KUKA KRL program: EPS_2_25252_SD5A_A_20250910061727.src

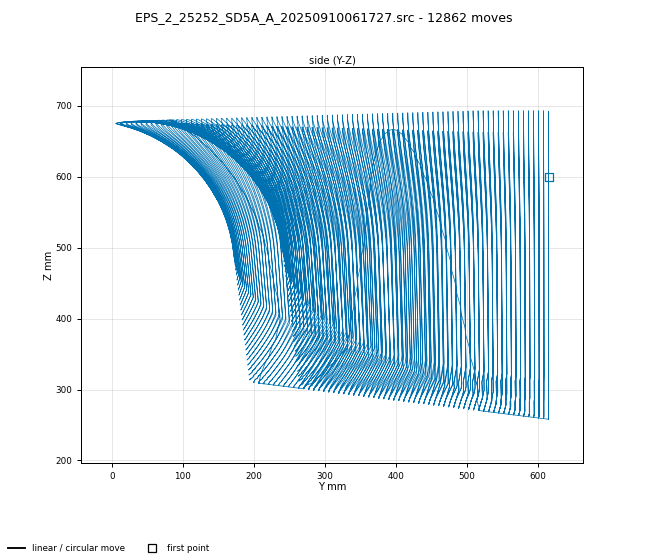
[picture p0: tool path of EPS_2_25252_SD5A_A_20250910061727.src, 12862 of 12864 moves have a stored position in this frame; points joined in program order, loops and branches not executed]
&ACCESS RVP
&REL 4
&COMMENT QRS 19112012
&PARAM EDITMASK = *
DEF PART()
EXT BAS (BAS_COMMAND :IN,REAL :IN )
INT I
BAS (#INITMOV,0 )

;KUKA QRS Post kuka4.cps  Date:22-06-2017 !

File_ID=2838

QRS_PRE_INIT()

;Init var - Until changes are made in qrs_pre_init
Outlet_Square_prg=0
Inlet_1_Square_prg=0
Inlet_2_Square_prg=0
Inlet_3_Square_prg=0
Inlet_4_Square_prg=0
Inlet_5_Square_prg=0

Outlet_1={X 0.000, Y 512.630, Z 510.000, B 0.000, E1 0.000 }
Inlet_1={X 0.000, Y 514.870, Z 480.000, B 0.000, E1 167.000 }
Outlet_1_type=366
Inlet_1_type=366
;QRS#1=Sidecore dimensions
;QRS#2=375-15" PVC SDR 35
;QRS#3=375-15" PVC SDR 35
;QRS#4=
;QRS#5=
;QRS#6=
;QRS#7=
;QRS#8=
;QRS#9=20Y PSX
;QRS#10=20Y PSX
;QRS#11=
;QRS#12=
;QRS#13=
;QRS#14=
;QRS#15=
;QRS#16=1220x127x991 3,25'
;QRS#17=EPS Height
;QRS#18=693
;QRS#19=*
;QRS#20= UPDATED VERSION 22-06-2017
;QRS#21=*
Outlet_Square=0250
Inlet_1_Square=0250
Inlet_2_Square=0
Inlet_3_Square=0
Inlet_4_Square=0
Inlet_5_Square=0
Mill_Square=1
Outlet_Square_Prg=252
Inlet_1_Square_prg=252

QRS_INIT()

$ADVANCE=5

; T1
PTP {E1 173.62,E2 173.62}
PTP {X 0,Y 615.5,A -85,B 0,C 180,E1 173.62,E2 173.62,E3 0,E4 0,E5 0,E6 0}
QRS_SPEED_INIT()
LIN {X 0,Y 615.5,Z 600,A -85,B 0,C 180,E1 173.62,E2 173.62,E3 0,E4 0,E5 0,E6 0} C_VEL
LIN {X 0,Y 615.5,Z 268.19,A -85,B 0,C 180,E1 173.62,E2 173.62} C_VEL
LIN {X 0,Y 615.5,Z 260.011,A -85,B 0,C 180,E1 173.62,E2 173.62} C_VEL
LIN {X 0,Y 615.475,Z 258.011,A -85,B 0,C 180,E1 173.434,E2 173.434} C_VEL
LIN {X 0,Y 615.437,Z 258.007,A -85,B 0,C 180,E1 170.8,E2 170.8} C_VEL
LIN {X 0,Y 615.481,Z 258.003,A -85,B 0,C 180,E1 168.139,E2 168.139} C_VEL
LIN {X 0,Y 615.462,Z 258.011,A -85,B 0,C 180,E1 165.45,E2 165.45} C_VEL
LIN {X 0,Y 615.455,Z 258.011,A -85,B 0,C 180,E1 163.412,E2 163.412} C_VEL
LIN {X 0,Y 615.445,Z 258.011,A -85,B 0,C 180,E1 161.352,E2 161.352} C_VEL
LIN {X 0,Y 615.436,Z 258.011,A -85,B 0,C 180,E1 159.267,E2 159.267} C_VEL
LIN {X 0,Y 615.426,Z 258.011,A -85,B 0,C 180,E1 157.153,E2 157.153} C_VEL
LIN {X 0,Y 615.418,Z 258.011,A -85,B 0,C 180,E1 155.005,E2 155.005} C_VEL
LIN {X 0,Y 615.418,Z 258.011,A -85,B 0,C 180,E1 152.819,E2 152.819} C_VEL
LIN {X 0,Y 615.467,Z 258.011,A -85,B 0,C 180,E1 150.209,E2 150.209} C_VEL
LIN {X 0,Y 615.438,Z 258.012,A -85,B 0,C 180,E1 147.539,E2 147.539} C_VEL
LIN {X 0,Y 615.413,Z 258.012,A -85,B 0,C 180,E1 145.18,E2 145.18} C_VEL
LIN {X 0,Y 615.42,Z 258.012,A -85,B 0,C 180,E1 142.753,E2 142.753} C_VEL
LIN {X 0,Y 615.486,Z 258.009,A -85,B 0,C 180,E1 139.911,E2 139.911} C_VEL
LIN {X 0,Y 615.451,Z 258.009,A -85,B 0,C 180,E1 137.643,E2 137.643} C_VEL
LIN {X 0,Y 615.422,Z 258.01,A -85,B 0,C 180,E1 135.075,E2 135.075} C_VEL
LIN {X 0,Y 615.425,Z 258.009,A -85,B 0,C 180,E1 133.04,E2 133.04} C_VEL
LIN {X 0,Y 615.45,Z 258.011,A -85,B 0,C 180,E1 130.61,E2 130.61} C_VEL
LIN {X 0,Y 615.454,Z 258.005,A -85,B 0,C 180,E1 127.628,E2 127.628} C_VEL
LIN {X 0,Y 615.432,Z 258.012,A -85,B 0,C 180,E1 127.246,E2 127.246} C_VEL
LIN {X 0,Y 615.457,Z 282.781,A -85,B 0,C 180,E1 124.979,E2 124.979} C_VEL
LIN {X 0,Y 615.491,Z 489.244,A -85,B 0,C 180,E1 122.426,E2 122.426} C_VEL
LIN {X 0,Y 615.493,Z 505.497,A -85,B 0,C 180,E1 122.088,E2 122.088} C_VEL
LIN {X 0,Y 615.497,Z 521.955,A -85,B 0,C 180,E1 121.61,E2 121.61} C_VEL
LIN {X 0,Y 615.49,Z 537.997,A -85,B 0,C 180,E1 121.002,E2 121.002} C_VEL
LIN {X 0,Y 615.49,Z 551.97,A -85,B 0,C 180,E1 120.349,E2 120.349} C_VEL
LIN {X 0,Y 615.498,Z 566.878,A -85,B 0,C 180,E1 119.503,E2 119.503} C_VEL
LIN {X 0,Y 615.494,Z 580.891,A -85,B 0,C 180,E1 118.554,E2 118.554} C_VEL
LIN {X 0,Y 615.493,Z 594.61,A -85,B 0,C 180,E1 117.453,E2 117.453} C_VEL
LIN {X 0,Y 615.494,Z 607.149,A -85,B 0,C 180,E1 116.261,E2 116.261} C_VEL
LIN {X 0,Y 615.496,Z 618.457,A -85,B 0,C 180,E1 114.992,E2 114.992} C_VEL
LIN {X 0,Y 615.493,Z 627.669,A -85,B 0,C 180,E1 113.782,E2 113.782} C_VEL
LIN {X 0,Y 615.491,Z 636.834,A -85,B 0,C 180,E1 112.346,E2 112.346} C_VEL
LIN {X 0,Y 615.491,Z 643.498,A -85,B 0,C 180,E1 111.081,E2 111.081} C_VEL
LIN {X 0,Y 615.491,Z 649.613,A -85,B 0,C 180,E1 109.685,E2 109.685} C_VEL
LIN {X 0,Y 615.486,Z 653.438,A -85,B 0,C 180,E1 108.603,E2 108.603} C_VEL
LIN {X 0,Y 615.483,Z 657.237,A -85,B 0,C 180,E1 107.271,E2 107.271} C_VEL
LIN {X 0,Y 615.491,Z 659.946,A -85,B 0,C 180,E1 105.905,E2 105.905} C_VEL
LIN {X 0,Y 615.493,Z 661.669,A -85,B 0,C 180,E1 104.549,E2 104.549} C_VEL
LIN {X 0,Y 615.485,Z 662.336,A -85,B 0,C 180,E1 103.201,E2 103.201} C_VEL
LIN {X 0,Y 615.493,Z 662.022,A -85,B 0,C 180,E1 101.861,E2 101.861} C_VEL
LIN {X 0,Y 615.489,Z 660.742,A -85,B 0,C 180,E1 100.527,E2 100.527} C_VEL
LIN {X 0,Y 615.492,Z 658.451,A -85,B 0,C 180,E1 99.199,E2 99.199} C_VEL
LIN {X 0,Y 615.496,Z 655.195,A -85,B 0,C 180,E1 97.876,E2 97.876} C_VEL
LIN {X 0,Y 615.488,Z 650.852,A -85,B 0,C 180,E1 96.557,E2 96.557} C_VEL
LIN {X 0,Y 615.492,Z 645.49,A -85,B 0,C 180,E1 95.241,E2 95.241} C_VEL
LIN {X 0,Y 615.488,Z 637.049,A -85,B 0,C 180,E1 93.601,E2 93.601} C_VEL
LIN {X 0,Y 615.488,Z 628.759,A -85,B 0,C 180,E1 92.291,E2 92.291} C_VEL
LIN {X 0,Y 615.493,Z 618.969,A -85,B 0,C 180,E1 90.981,E2 90.981} C_VEL
LIN {X 0,Y 615.491,Z 607.385,A -85,B 0,C 180,E1 89.673,E2 89.673} C_VEL
LIN {X 0,Y 615.494,Z 595.424,A -85,B 0,C 180,E1 88.528,E2 88.528} C_VEL
LIN {X 0,Y 615.496,Z 582.372,A -85,B 0,C 180,E1 87.464,E2 87.464} C_VEL
LIN {X 0,Y 615.498,Z 569.42,A -85,B 0,C 180,E1 86.563,E2 86.563} C_VEL
LIN {X 0,Y 615.498,Z 555.382,A -85,B 0,C 180,E1 85.744,E2 85.744} C_VEL
LIN {X 0,Y 615.498,Z 540.224,A -85,B 0,C 180,E1 85.005,E2 85.005} C_VEL
LIN {X 0,Y 615.498,Z 524.623,A -85,B 0,C 180,E1 84.389,E2 84.389} C_VEL
LIN {X 0,Y 615.497,Z 508.547,A -85,B 0,C 180,E1 83.896,E2 83.896} C_VEL
LIN {X 0,Y 615.489,Z 491.531,A -85,B 0,C 180,E1 83.526,E2 83.526} C_VEL
LIN {X 0,Y 615.495,Z 466.17,A -85,B 0,C 180,E1 83.185,E2 83.185} C_VEL
LIN {X 0,Y 615.461,Z 282.717,A -85,B 0,C 180,E1 80.925,E2 80.925} C_VEL
LIN {X 0,Y 615.44,Z 258.005,A -85,B 0,C 180,E1 78.66,E2 78.66} C_VEL
LIN {X 0,Y 615.49,Z 258.002,A -85,B 0,C 180,E1 76.068,E2 76.068} C_VEL
LIN {X 0,Y 615.462,Z 258.011,A -85,B 0,C 180,E1 73.413,E2 73.413} C_VEL
LIN {X 0,Y 615.453,Z 258.011,A -85,B 0,C 180,E1 71.353,E2 71.353} C_VEL
LIN {X 0,Y 615.443,Z 258.01,A -85,B 0,C 180,E1 69.268,E2 69.268} C_VEL
LIN {X 0,Y 615.434,Z 258.01,A -85,B 0,C 180,E1 67.153,E2 67.153} C_VEL
LIN {X 0,Y 615.426,Z 258.01,A -85,B 0,C 180,E1 65.006,E2 65.006} C_VEL
LIN {X 0,Y 615.424,Z 258.009,A -85,B 0,C 180,E1 62.82,E2 62.82} C_VEL
LIN {X 0,Y 615.469,Z 258.008,A -85,B 0,C 180,E1 60.209,E2 60.209} C_VEL
LIN {X 0,Y 615.45,Z 258.012,A -85,B 0,C 180,E1 57.54,E2 57.54} C_VEL
LIN {X 0,Y 615.418,Z 258.012,A -85,B 0,C 180,E1 55.18,E2 55.18} C_VEL
LIN {X 0,Y 615.417,Z 258.012,A -85,B 0,C 180,E1 52.753,E2 52.753} C_VEL
LIN {X 0,Y 615.488,Z 258.012,A -85,B 0,C 180,E1 49.912,E2 49.912} C_VEL
LIN {X 0,Y 615.447,Z 258.012,A -85,B 0,C 180,E1 47.644,E2 47.644} C_VEL
LIN {X 0,Y 615.413,Z 258.012,A -85,B 0,C 180,E1 45.076,E2 45.076} C_VEL
LIN {X 0,Y 615.414,Z 258.011,A -85,B 0,C 180,E1 43.04,E2 43.04} C_VEL
LIN {X 0,Y 615.417,Z 258.011,A -85,B 0,C 180,E1 41.087,E2 41.087} C_VEL
LIN {X 0,Y 615.421,Z 258.011,A -85,B 0,C 180,E1 38.91,E2 38.91} C_VEL
LIN {X 0,Y 615.459,Z 258.012,A -85,B 0,C 180,E1 36.427,E2 36.427} C_VEL
LIN {X 0,Y 615.442,Z 258.008,A -85,B 0,C 180,E1 33.528,E2 33.528} C_VEL
LIN {X 0,Y 615.427,Z 258.009,A -85,B 0,C 180,E1 31.077,E2 31.077} C_VEL
LIN {X 0,Y 615.445,Z 258.011,A -85,B 0,C 180,E1 28.661,E2 28.661} C_VEL
LIN {X 0,Y 615.463,Z 258.004,A -85,B 0,C 180,E1 25.717,E2 25.717} C_VEL
LIN {X 0,Y 615.449,Z 258.005,A -85,B 0,C 180,E1 23.558,E2 23.558} C_VEL
LIN {X 0,Y 615.443,Z 258.005,A -85,B 0,C 180,E1 21.434,E2 21.434} C_VEL
LIN {X 0,Y 615.44,Z 258.005,A -85,B 0,C 180,E1 19.34,E2 19.34} C_VEL
LIN {X 0,Y 615.44,Z 258.006,A -85,B 0,C 180,E1 17.272,E2 17.272} C_VEL
LIN {X 0,Y 615.482,Z 258.011,A -85,B 0,C 180,E1 14.55,E2 14.55} C_VEL
LIN {X 0,Y 615.482,Z 258,A -85,B 0,C 180,E1 11.861,E2 11.861} C_VEL
LIN {X 0,Y 615.447,Z 258.006,A -85,B 0,C 180,E1 9.2,E2 9.2} C_VEL
LIN {X 0,Y 615.491,Z 258.013,A -85,B 0,C 180,E1 6.557,E2 6.557} C_VEL
LIN {X 0,Y 615.484,Z 257.999,A -85,B 0,C 180,E1 3.929,E2 3.929} C_VEL
LIN {X 0,Y 615.453,Z 258.004,A -85,B 0,C 180,E1 1.309,E2 1.309} C_VEL
LIN {X 0,Y 615.489,Z 258.011,A -85,B 0,C 180,E1 -1.308,E2 -1.308} C_VEL
LIN {X 0,Y 615.49,Z 257.998,A -85,B 0,C 180,E1 -3.928,E2 -3.928} C_VEL
LIN {X 0,Y 615.46,Z 258.002,A -85,B 0,C 180,E1 -6.557,E2 -6.557} C_VEL
LIN {X 0,Y 615.488,Z 258.011,A -85,B 0,C 180,E1 -9.198,E2 -9.198} C_VEL
LIN {X 0,Y 615.493,Z 257.997,A -85,B 0,C 180,E1 -11.86,E2 -11.86} C_VEL
LIN {X 0,Y 615.465,Z 258.002,A -85,B 0,C 180,E1 -14.549,E2 -14.549} C_VEL
LIN {X 0,Y 615.493,Z 258.012,A -85,B 0,C 180,E1 -17.27,E2 -17.27} C_VEL
LIN {X 0,Y 615.488,Z 257.995,A -85,B 0,C 180,E1 -20.032,E2 -20.032} C_VEL
LIN {X 0,Y 615.477,Z 258.007,A -85,B 0,C 180,E1 -22.845,E2 -22.845} C_VEL
LIN {X 0,Y 615.481,Z 257.999,A -85,B 0,C 180,E1 -25.716,E2 -25.716} C_VEL
LIN {X 0,Y 615.474,Z 258.001,A -85,B 0,C 180,E1 -28.448,E2 -28.448} C_VEL
LIN {X 0,Y 615.484,Z 258.015,A -85,B 0,C 180,E1 -31.085,E2 -31.085} C_VEL
LIN {X 0,Y 615.493,Z 257.993,A -85,B 0,C 180,E1 -34.021,E2 -34.021} C_VEL
LIN {X 0,Y 615.488,Z 258.014,A -85,B 0,C 180,E1 -36.937,E2 -36.937} C_VEL
LIN {X 0,Y 615.478,Z 257.998,A -85,B 0,C 180,E1 -39.751,E2 -39.751} C_VEL
LIN {X 0,Y 615.482,Z 258,A -85,B 0,C 180,E1 -42.353,E2 -42.353} C_VEL
LIN {X 0,Y 615.484,Z 258.009,A -85,B 0,C 180,E1 -45.069,E2 -45.069} C_VEL
LIN {X 0,Y 615.489,Z 257.995,A -85,B 0,C 180,E1 -47.919,E2 -47.919} C_VEL
LIN {X 0,Y 615.487,Z 258.01,A -85,B 0,C 180,E1 -50.938,E2 -50.938} C_VEL
LIN {X 0,Y 615.469,Z 258,A -85,B 0,C 180,E1 -53.574,E2 -53.574} C_VEL
LIN {X 0,Y 615.488,Z 258.006,A -85,B 0,C 180,E1 -56.465,E2 -56.465} C_VEL
LIN {X 0,Y 615.469,Z 258.007,A -85,B 0,C 180,E1 -59.079,E2 -59.079} C_VEL
LIN {X 0,Y 615.464,Z 258,A -85,B 0,C 180,E1 -61.553,E2 -61.553} C_VEL
LIN {X 0,Y 615.465,Z 258.184,A -85,B 0,C 180,E1 -63.601,E2 -63.601} C_VEL
LIN {X 0,Y 615.476,Z 290.167,A -85,B 0,C 180,E1 -66.217,E2 -66.217} C_VEL
LIN {X 0,Y 615.493,Z 312.012,A -85,B 0,C 180,E1 -67.974,E2 -67.974} C_VEL
LIN {X 0,Y 615.491,Z 519.433,A -85,B 0,C 180,E1 -70.532,E2 -70.532} C_VEL
LIN {X 0,Y 615.493,Z 535.998,A -85,B 0,C 180,E1 -70.879,E2 -70.879} C_VEL
LIN {X 0,Y 615.493,Z 550.934,A -85,B 0,C 180,E1 -71.311,E2 -71.311} C_VEL
LIN {X 0,Y 615.491,Z 566.349,A -85,B 0,C 180,E1 -71.881,E2 -71.881} C_VEL
LIN {X 0,Y 615.493,Z 581.006,A -85,B 0,C 180,E1 -72.558,E2 -72.558} C_VEL
LIN {X 0,Y 615.5,Z 594.837,A -85,B 0,C 180,E1 -73.328,E2 -73.328} C_VEL
LIN {X 0,Y 615.499,Z 609.038,A -85,B 0,C 180,E1 -74.265,E2 -74.265} C_VEL
LIN {X 0,Y 615.495,Z 622.093,A -85,B 0,C 180,E1 -75.282,E2 -75.282} C_VEL
LIN {X 0,Y 615.494,Z 633.214,A -85,B 0,C 180,E1 -76.294,E2 -76.294} C_VEL
LIN {X 0,Y 615.493,Z 644.291,A -85,B 0,C 180,E1 -77.47,E2 -77.47} C_VEL
LIN {X 0,Y 615.494,Z 653.767,A -85,B 0,C 180,E1 -78.64,E2 -78.64} C_VEL
LIN {X 0,Y 615.496,Z 662.964,A -85,B 0,C 180,E1 -79.972,E2 -79.972} C_VEL
LIN {X 0,Y 615.489,Z 671.502,A -85,B 0,C 180,E1 -81.463,E2 -81.463} C_VEL
LIN {X 0,Y 615.491,Z 678.982,A -85,B 0,C 180,E1 -83.102,E2 -83.102} C_VEL
LIN {X 0,Y 615.492,Z 684.741,A -85,B 0,C 180,E1 -84.759,E2 -84.759} C_VEL
LIN {X 0,Y 615.494,Z 688.076,A -85,B 0,C 180,E1 -86.072,E2 -86.072} C_VEL
LIN {X 0,Y 615.485,Z 690.504,A -85,B 0,C 180,E1 -87.382,E2 -87.382} C_VEL
LIN {X 0,Y 615.488,Z 691.87,A -85,B 0,C 180,E1 -88.691,E2 -88.691} C_VEL
LIN {X 0,Y 615.489,Z 692.39,A -85,B 0,C 180,E1 -90,E2 -90} C_VEL
LIN {X 0,Y 615.488,Z 691.87,A -85,B 0,C 180,E1 -91.309,E2 -91.309} C_VEL
LIN {X 0,Y 615.485,Z 690.504,A -85,B 0,C 180,E1 -92.618,E2 -92.618} C_VEL
LIN {X 0,Y 615.494,Z 688.076,A -85,B 0,C 180,E1 -93.929,E2 -93.929} C_VEL
LIN {X 0,Y 615.492,Z 684.741,A -85,B 0,C 180,E1 -95.241,E2 -95.241} C_VEL
LIN {X 0,Y 615.491,Z 678.982,A -85,B 0,C 180,E1 -96.898,E2 -96.898} C_VEL
LIN {X 0,Y 615.489,Z 671.501,A -85,B 0,C 180,E1 -98.537,E2 -98.537} C_VEL
LIN {X 0,Y 615.496,Z 662.963,A -85,B 0,C 180,E1 -100.028,E2 -100.028} C_VEL
LIN {X 0,Y 615.494,Z 653.765,A -85,B 0,C 180,E1 -101.36,E2 -101.36} C_VEL
LIN {X 0,Y 615.495,Z 644.29,A -85,B 0,C 180,E1 -102.53,E2 -102.53} C_VEL
LIN {X 0,Y 615.494,Z 633.212,A -85,B 0,C 180,E1 -103.706,E2 -103.706} C_VEL
LIN {X 0,Y 615.495,Z 621.113,A -85,B 0,C 180,E1 -104.803,E2 -104.803} C_VEL
LIN {X 0,Y 615.498,Z 606.706,A -85,B 0,C 180,E1 -105.905,E2 -105.905} C_VEL
LIN {X 0,Y 615.497,Z 592.012,A -85,B 0,C 180,E1 -106.843,E2 -106.843} C_VEL
LIN {X 0,Y 615.49,Z 577.507,A -85,B 0,C 180,E1 -107.613,E2 -107.613} C_VEL
LIN {X 0,Y 615.49,Z 562.245,A -85,B 0,C 180,E1 -108.282,E2 -108.282} C_VEL
LIN {X 0,Y 615.49,Z 546.989,A -85,B 0,C 180,E1 -108.819,E2 -108.819} C_VEL
LIN {X 0,Y 615.497,Z 530.513,A -85,B 0,C 180,E1 -109.251,E2 -109.251} C_VEL
LIN {X 0,Y 615.49,Z 514.919,A -85,B 0,C 180,E1 -109.533,E2 -109.533} C_VEL
LIN {X 0,Y 615.493,Z 312.01,A -85,B 0,C 180,E1 -112.026,E2 -112.026} C_VEL
LIN {X 0,Y 615.458,Z 276.401,A -85,B 0,C 180,E1 -114.903,E2 -114.903} C_VEL
LIN {X 0,Y 615.464,Z 258,A -85,B 0,C 180,E1 -116.422,E2 -116.422} C_VEL
LIN {X 0,Y 615.461,Z 258.003,A -85,B 0,C 180,E1 -118.66,E2 -118.66} C_VEL
LIN {X 0,Y 615.481,Z 258.01,A -85,B 0,C 180,E1 -121.085,E2 -121.085} C_VEL
LIN {X 0,Y 615.493,Z 257.995,A -85,B 0,C 180,E1 -124.022,E2 -124.022} C_VEL
LIN {X 0,Y 615.478,Z 258.008,A -85,B 0,C 180,E1 -126.936,E2 -126.936} C_VEL
LIN {X 0,Y 615.483,Z 257.999,A -85,B 0,C 180,E1 -129.751,E2 -129.751} C_VEL
LIN {X 0,Y 615.475,Z 257.999,A -85,B 0,C 180,E1 -132.354,E2 -132.354} C_VEL
LIN {X 0,Y 615.493,Z 258.014,A -85,B 0,C 180,E1 -135.068,E2 -135.068} C_VEL
LIN {X 0,Y 615.49,Z 257.995,A -85,B 0,C 180,E1 -137.92,E2 -137.92} C_VEL
LIN {X 0,Y 615.482,Z 257.997,A -85,B 0,C 180,E1 -140.25,E2 -140.25} C_VEL
LIN {X 0,Y 615.491,Z 258.011,A -85,B 0,C 180,E1 -143.063,E2 -143.063} C_VEL
LIN {X 0,Y 615.491,Z 257.994,A -85,B 0,C 180,E1 -145.979,E2 -145.979} C_VEL
LIN {X 0,Y 615.486,Z 258.015,A -85,B 0,C 180,E1 -148.915,E2 -148.915} C_VEL
LIN {X 0,Y 615.471,Z 258,A -85,B 0,C 180,E1 -151.553,E2 -151.553} C_VEL
LIN {X 0,Y 615.486,Z 258,A -85,B 0,C 180,E1 -154.285,E2 -154.285} C_VEL
LIN {X 0,Y 615.486,Z 258.004,A -85,B 0,C 180,E1 -156.444,E2 -156.444} C_VEL
LIN {X 0,Y 615.465,Z 258.005,A -85,B 0,C 180,E1 -159.269,E2 -159.269} C_VEL
LIN {X 0,Y 615.493,Z 257.996,A -85,B 0,C 180,E1 -162.044,E2 -162.044} C_VEL
LIN {X 0,Y 615.484,Z 258.012,A -85,B 0,C 180,E1 -164.774,E2 -164.774} C_VEL
LIN {X 0,Y 615.459,Z 258.002,A -85,B 0,C 180,E1 -167.47,E2 -167.47} C_VEL
LIN {X 0,Y 615.493,Z 258,A -85,B 0,C 180,E1 -170.138,E2 -170.138} C_VEL
LIN {X 0,Y 615.474,Z 258.01,A -85,B 0,C 180,E1 -172.785,E2 -172.785} C_VEL
LIN {X 0,Y 615.452,Z 258.003,A -85,B 0,C 180,E1 -175.416,E2 -175.416} C_VEL
LIN {X 0,Y 615.498,Z 257.999,A -85,B 0,C 180,E1 -178.037,E2 -178.037} C_VEL
LIN {X 0,Y 615.474,Z 258.011,A -85,B 0,C 180,E1 -180.655,E2 -180.655} C_VEL
LIN {X 0,Y 615.443,Z 258.005,A -85,B 0,C 180,E1 -183.274,E2 -183.274} C_VEL
LIN {X 0,Y 615.485,Z 258.001,A -85,B 0,C 180,E1 -185.899,E2 -185.899} C_VEL
LIN {X 0,Y 615.475,Z 258.011,A -85,B 0,C 180,E1 -186.566,E2 -186.566} C_VEL
LIN {X 0,Y 614.772,Z 258.153,A -85,B 0,C 180,E1 -187.112,E2 -187.112} C_VEL
LIN {X 0,Y 611.917,Z 258.573,A -85,B 0,C 180,E1 -187.998,E2 -187.998} C_VEL
LIN {X 0,Y 609.53,Z 258.879,A -85,B 0,C 180,E1 -188.711,E2 -188.711} C_VEL
LIN {X 0,Y 608.51,Z 258.994,A -85,B 0,C 180,E1 -189.26,E2 -189.26} C_VEL
LIN {X 0,Y 608.428,Z 259.003,A -85,B 0,C 180,E1 -189.446,E2 -189.446} C_VEL
LIN {X 0,Y 608.455,Z 259.005,A -85,B 0,C 180,E1 -192,E2 -192} C_VEL
LIN {X 0,Y 608.417,Z 259.007,A -85,B 0,C 180,E1 -194.722,E2 -194.722} C_VEL
LIN {X 0,Y 608.419,Z 259.006,A -85,B 0,C 180,E1 -196.785,E2 -196.785} C_VEL
LIN {X 0,Y 608.421,Z 259.005,A -85,B 0,C 180,E1 -199.572,E2 -199.572} C_VEL
LIN {X 0,Y 608.433,Z 259.007,A -85,B 0,C 180,E1 -202.47,E2 -202.47} C_VEL
LIN {X 0,Y 608.424,Z 259.007,A -85,B 0,C 180,E1 -204.573,E2 -204.573} C_VEL
LIN {X 0,Y 608.403,Z 259.006,A -85,B 0,C 180,E1 -207.193,E2 -207.193} C_VEL
LIN {X 0,Y 608.455,Z 259.009,A -85,B 0,C 180,E1 -209.969,E2 -209.969} C_VEL
LIN {X 0,Y 608.407,Z 259.006,A -85,B 0,C 180,E1 -212.883,E2 -212.883} C_VEL
LIN {X 0,Y 608.398,Z 259.008,A -85,B 0,C 180,E1 -215.281,E2 -215.281} C_VEL
LIN {X 0,Y 608.423,Z 259.009,A -85,B 0,C 180,E1 -218.235,E2 -218.235} C_VEL
LIN {X 0,Y 608.437,Z 259.006,A -85,B 0,C 180,E1 -220.327,E2 -220.327} C_VEL
LIN {X 0,Y 608.425,Z 259.007,A -85,B 0,C 180,E1 -222.33,E2 -222.33} C_VEL
LIN {X 0,Y 608.404,Z 259.006,A -85,B 0,C 180,E1 -224.801,E2 -224.801} C_VEL
LIN {X 0,Y 608.397,Z 259.007,A -85,B 0,C 180,E1 -227.035,E2 -227.035} C_VEL
LIN {X 0,Y 608.399,Z 259.007,A -85,B 0,C 180,E1 -228.819,E2 -228.819} C_VEL
LIN {X 0,Y 608.41,Z 259.01,A -85,B 0,C 180,E1 -231.407,E2 -231.407} C_VEL
LIN {X 0,Y 608.448,Z 259.144,A -85,B 0,C 180,E1 -232.562,E2 -232.562} C_VEL
LIN {X 0,Y 608.699,Z 265.928,A -85,B 0,C 180,E1 -233.206,E2 -233.206} C_VEL
LIN {X 0,Y 608.688,Z 283.12,A -85,B 0,C 180,E1 -234.776,E2 -234.776} C_VEL
LIN {X 0,Y 608.886,Z 299.347,A -85,B 0,C 180,E1 -234.986,E2 -234.986} C_VEL
LIN {X 0,Y 608.795,Z 489.212,A -85,B 0,C 180,E1 -237.351,E2 -237.351} C_VEL
LIN {X 0,Y 608.774,Z 505.767,A -85,B 0,C 180,E1 -237.699,E2 -237.699} C_VEL
LIN {X 0,Y 608.739,Z 521.663,A -85,B 0,C 180,E1 -238.165,E2 -238.165} C_VEL
LIN {X 0,Y 608.695,Z 537.166,A -85,B 0,C 180,E1 -238.752,E2 -238.752} C_VEL
LIN {X 0,Y 608.651,Z 552.299,A -85,B 0,C 180,E1 -239.465,E2 -239.465} C_VEL
LIN {X 0,Y 608.632,Z 567.204,A -85,B 0,C 180,E1 -240.324,E2 -240.324} C_VEL
LIN {X 0,Y 608.591,Z 580.323,A -85,B 0,C 180,E1 -241.221,E2 -241.221} C_VEL
LIN {X 0,Y 608.545,Z 593.768,A -85,B 0,C 180,E1 -242.3,E2 -242.3} C_VEL
LIN {X 0,Y 608.523,Z 605.625,A -85,B 0,C 180,E1 -243.414,E2 -243.414} C_VEL
LIN {X 0,Y 608.478,Z 616.052,A -85,B 0,C 180,E1 -244.554,E2 -244.554} C_VEL
LIN {X 0,Y 608.477,Z 626.718,A -85,B 0,C 180,E1 -245.927,E2 -245.927} C_VEL
LIN {X 0,Y 608.464,Z 635.273,A -85,B 0,C 180,E1 -247.236,E2 -247.236} C_VEL
LIN {X 0,Y 608.455,Z 643.098,A -85,B 0,C 180,E1 -248.663,E2 -248.663} C_VEL
LIN {X 0,Y 608.433,Z 649.462,A -85,B 0,C 180,E1 -250.077,E2 -250.077} C_VEL
LIN {X 0,Y 608.423,Z 653.828,A -85,B 0,C 180,E1 -251.299,E2 -251.299} C_VEL
LIN {X 0,Y 608.41,Z 657.363,A -85,B 0,C 180,E1 -252.522,E2 -252.522} C_VEL
LIN {X 0,Y 608.428,Z 660.267,A -85,B 0,C 180,E1 -253.905,E2 -253.905} C_VEL
LIN {X 0,Y 608.416,Z 662.146,A -85,B 0,C 180,E1 -255.278,E2 -255.278} C_VEL
LIN {X 0,Y 608.431,Z 662.911,A -85,B 0,C 180,E1 -256.643,E2 -256.643} C_VEL
LIN {X 0,Y 608.437,Z 662.738,A -85,B 0,C 180,E1 -258,E2 -258} C_VEL
LIN {X 0,Y 608.43,Z 661.512,A -85,B 0,C 180,E1 -259.349,E2 -259.349} C_VEL
LIN {X 0,Y 608.419,Z 659.338,A -85,B 0,C 180,E1 -260.693,E2 -260.693} C_VEL
LIN {X 0,Y 608.42,Z 656.121,A -85,B 0,C 180,E1 -262.032,E2 -262.032} C_VEL
LIN {X 0,Y 608.448,Z 651.761,A -85,B 0,C 180,E1 -263.397,E2 -263.397} C_VEL
LIN {X 0,Y 608.456,Z 646.54,A -85,B 0,C 180,E1 -264.698,E2 -264.698} C_VEL
LIN {X 0,Y 608.434,Z 639.993,A -85,B 0,C 180,E1 -266.026,E2 -266.026} C_VEL
LIN {X 0,Y 608.46,Z 632.217,A -85,B 0,C 180,E1 -267.352,E2 -267.352} C_VEL
LIN {X 0,Y 608.478,Z 622.95,A -85,B 0,C 180,E1 -268.676,E2 -268.676} C_VEL
LIN {X 0,Y 608.486,Z 611.978,A -85,B 0,C 180,E1 -270,E2 -270} C_VEL
LIN {X 0,Y 608.519,Z 600.706,A -85,B 0,C 180,E1 -271.158,E2 -271.158} C_VEL
LIN {X 0,Y 608.558,Z 587.484,A -85,B 0,C 180,E1 -272.316,E2 -272.316} C_VEL
LIN {X 0,Y 608.612,Z 574.126,A -85,B 0,C 180,E1 -273.31,E2 -273.31} C_VEL
LIN {X 0,Y 608.638,Z 559.633,A -85,B 0,C 180,E1 -274.221,E2 -274.221} C_VEL
LIN {X 0,Y 608.673,Z 545.387,A -85,B 0,C 180,E1 -274.968,E2 -274.968} C_VEL
LIN {X 0,Y 608.73,Z 529.827,A -85,B 0,C 180,E1 -275.632,E2 -275.632} C_VEL
LIN {X 0,Y 608.763,Z 513.799,A -85,B 0,C 180,E1 -276.172,E2 -276.172} C_VEL
LIN {X 0,Y 608.789,Z 497.872,A -85,B 0,C 180,E1 -276.575,E2 -276.575} C_VEL
LIN {X 0,Y 608.805,Z 481.487,A -85,B 0,C 180,E1 -276.851,E2 -276.851} C_VEL
LIN {X 0,Y 608.878,Z 285.382,A -85,B 0,C 180,E1 -279.279,E2 -279.279} C_VEL
LIN {X 0,Y 608.668,Z 282.6,A -85,B 0,C 180,E1 -279.345,E2 -279.345} C_VEL
LIN {X 0,Y 608.696,Z 261.258,A -85,B 0,C 180,E1 -281.32,E2 -281.32} C_VEL
LIN {X 0,Y 608.442,Z 259.004,A -85,B 0,C 180,E1 -281.556,E2 -281.556} C_VEL
LIN {X 0,Y 608.475,Z 259.003,A -85,B 0,C 180,E1 -284.037,E2 -284.037} C_VEL
LIN {X 0,Y 608.424,Z 259.006,A -85,B 0,C 180,E1 -286.785,E2 -286.785} C_VEL
LIN {X 0,Y 608.424,Z 259.005,A -85,B 0,C 180,E1 -289.571,E2 -289.571} C_VEL
LIN {X 0,Y 608.439,Z 259.009,A -85,B 0,C 180,E1 -292.407,E2 -292.407} C_VEL
LIN {X 0,Y 608.43,Z 259.007,A -85,B 0,C 180,E1 -294.572,E2 -294.572} C_VEL
LIN {X 0,Y 608.408,Z 259.005,A -85,B 0,C 180,E1 -297.193,E2 -297.193} C_VEL
LIN {X 0,Y 608.46,Z 259.007,A -85,B 0,C 180,E1 -299.969,E2 -299.969} C_VEL
LIN {X 0,Y 608.414,Z 259.005,A -85,B 0,C 180,E1 -302.882,E2 -302.882} C_VEL
LIN {X 0,Y 608.399,Z 259.007,A -85,B 0,C 180,E1 -305.281,E2 -305.281} C_VEL
LIN {X 0,Y 608.424,Z 259.01,A -85,B 0,C 180,E1 -308.234,E2 -308.234} C_VEL
LIN {X 0,Y 608.436,Z 259.007,A -85,B 0,C 180,E1 -310.327,E2 -310.327} C_VEL
LIN {X 0,Y 608.421,Z 259.008,A -85,B 0,C 180,E1 -312.329,E2 -312.329} C_VEL
LIN {X 0,Y 608.396,Z 259.007,A -85,B 0,C 180,E1 -314.801,E2 -314.801} C_VEL
LIN {X 0,Y 608.387,Z 259.008,A -85,B 0,C 180,E1 -317.034,E2 -317.034} C_VEL
LIN {X 0,Y 608.389,Z 259.008,A -85,B 0,C 180,E1 -318.817,E2 -318.817} C_VEL
LIN {X 0,Y 608.404,Z 259.006,A -85,B 0,C 180,E1 -320.71,E2 -320.71} C_VEL
LIN {X 0,Y 608.394,Z 259.007,A -85,B 0,C 180,E1 -323.08,E2 -323.08} C_VEL
LIN {X 0,Y 608.441,Z 259.006,A -85,B 0,C 180,E1 -325.528,E2 -325.528} C_VEL
LIN {X 0,Y 608.455,Z 259.008,A -85,B 0,C 180,E1 -327.904,E2 -327.904} C_VEL
LIN {X 0,Y 608.456,Z 259.002,A -85,B 0,C 180,E1 -330.219,E2 -330.219} C_VEL
LIN {X 0,Y 608.412,Z 259.005,A -85,B 0,C 180,E1 -332.805,E2 -332.805} C_VEL
LIN {X 0,Y 608.436,Z 259.008,A -85,B 0,C 180,E1 -335.428,E2 -335.428} C_VEL
LIN {X 0,Y 608.448,Z 259.002,A -85,B 0,C 180,E1 -338.307,E2 -338.307} C_VEL
LIN {X 0,Y 608.439,Z 259.004,A -85,B 0,C 180,E1 -341.129,E2 -341.129} C_VEL
LIN {X 0,Y 608.46,Z 259.004,A -85,B 0,C 180,E1 -343.906,E2 -343.906} C_VEL
LIN {X 0,Y 608.433,Z 259.002,A -85,B 0,C 180,E1 -346.642,E2 -346.642} C_VEL
LIN {X 0,Y 608.456,Z 259.006,A -85,B 0,C 180,E1 -349.35,E2 -349.35} C_VEL
LIN {X 0,Y 608.475,Z 259,A -85,B 0,C 180,E1 -352.033,E2 -352.033} C_VEL
LIN {X 0,Y 608.435,Z 259.002,A -85,B 0,C 180,E1 -354.697,E2 -354.697} C_VEL
LIN {X 0,Y 608.481,Z 259.005,A -85,B 0,C 180,E1 -357.352,E2 -357.352} C_VEL
LIN {X 0,Y 608.477,Z 258.998,A -85,B 0,C 180,E1 -360,E2 -360} C_VEL
LIN {X 0,Y 608.451,Z 259.001,A -85,B 0,C 180,E1 -362.648,E2 -362.648} C_VEL
LIN {X 0,Y 608.468,Z 259.008,A -85,B 0,C 180,E1 -365.301,E2 -365.301} C_VEL
LIN {X 0,Y 608.479,Z 258.998,A -85,B 0,C 180,E1 -367.967,E2 -367.967} C_VEL
LIN {X 0,Y 608.444,Z 259.002,A -85,B 0,C 180,E1 -370.65,E2 -370.65} C_VEL
LIN {X 0,Y 608.471,Z 259.007,A -85,B 0,C 180,E1 -373.356,E2 -373.356} C_VEL
LIN {X 0,Y 608.457,Z 258.999,A -85,B 0,C 180,E1 -376.094,E2 -376.094} C_VEL
LIN {X 0,Y 608.449,Z 259.005,A -85,B 0,C 180,E1 -378.869,E2 -378.869} C_VEL
LIN {X 0,Y 608.467,Z 259,A -85,B 0,C 180,E1 -381.691,E2 -381.691} C_VEL
LIN {X 0,Y 608.451,Z 259.002,A -85,B 0,C 180,E1 -384.571,E2 -384.571} C_VEL
LIN {X 0,Y 608.483,Z 259.005,A -85,B 0,C 180,E1 -387.208,E2 -387.208} C_VEL
LIN {X 0,Y 608.468,Z 258.998,A -85,B 0,C 180,E1 -389.971,E2 -389.971} C_VEL
LIN {X 0,Y 608.451,Z 259.008,A -85,B 0,C 180,E1 -392.88,E2 -392.88} C_VEL
LIN {X 0,Y 608.439,Z 259.007,A -85,B 0,C 180,E1 -395.278,E2 -395.278} C_VEL
LIN {X 0,Y 608.467,Z 258.998,A -85,B 0,C 180,E1 -397.746,E2 -397.746} C_VEL
LIN {X 0,Y 608.454,Z 259.001,A -85,B 0,C 180,E1 -400.329,E2 -400.329} C_VEL
LIN {X 0,Y 608.453,Z 259.01,A -85,B 0,C 180,E1 -402.959,E2 -402.959} C_VEL
LIN {X 0,Y 608.456,Z 259,A -85,B 0,C 180,E1 -405.736,E2 -405.736} C_VEL
LIN {X 0,Y 608.461,Z 259.006,A -85,B 0,C 180,E1 -408.658,E2 -408.658} C_VEL
LIN {X 0,Y 608.462,Z 259,A -85,B 0,C 180,E1 -411.412,E2 -411.412} C_VEL
LIN {X 0,Y 608.46,Z 258.999,A -85,B 0,C 180,E1 -413.952,E2 -413.952} C_VEL
LIN {X 0,Y 608.466,Z 259.002,A -85,B 0,C 180,E1 -416.329,E2 -416.329} C_VEL
LIN {X 0,Y 608.459,Z 259.01,A -85,B 0,C 180,E1 -418.73,E2 -418.73} C_VEL
LIN {X 0,Y 608.453,Z 259.001,A -85,B 0,C 180,E1 -421.383,E2 -421.383} C_VEL
LIN {X 0,Y 608.449,Z 259.012,A -85,B 0,C 180,E1 -423.342,E2 -423.342} C_VEL
LIN {X 0,Y 608.824,Z 262.049,A -85,B 0,C 180,E1 -423.613,E2 -423.613} C_VEL
LIN {X 0,Y 608.729,Z 296.278,A -85,B 0,C 180,E1 -426.437,E2 -426.437} C_VEL
LIN {X 0,Y 608.713,Z 312.012,A -85,B 0,C 180,E1 -427.716,E2 -427.716} C_VEL
LIN {X 0,Y 608.9,Z 322.557,A -85,B 0,C 180,E1 -427.857,E2 -427.857} C_VEL
LIN {X 0,Y 608.795,Z 517.942,A -85,B 0,C 180,E1 -430.287,E2 -430.287} C_VEL
LIN {X 0,Y 608.796,Z 534.173,A -85,B 0,C 180,E1 -430.616,E2 -430.616} C_VEL
LIN {X 0,Y 608.737,Z 549.644,A -85,B 0,C 180,E1 -431.052,E2 -431.052} C_VEL
LIN {X 0,Y 608.711,Z 564.369,A -85,B 0,C 180,E1 -431.589,E2 -431.589} C_VEL
LIN {X 0,Y 608.678,Z 579.262,A -85,B 0,C 180,E1 -432.27,E2 -432.27} C_VEL
LIN {X 0,Y 608.616,Z 594.84,A -85,B 0,C 180,E1 -433.134,E2 -433.134} C_VEL
LIN {X 0,Y 608.579,Z 609.047,A -85,B 0,C 180,E1 -434.082,E2 -434.082} C_VEL
LIN {X 0,Y 608.556,Z 622.128,A -85,B 0,C 180,E1 -435.11,E2 -435.11} C_VEL
LIN {X 0,Y 608.528,Z 634.009,A -85,B 0,C 180,E1 -436.204,E2 -436.204} C_VEL
LIN {X 0,Y 608.49,Z 645.912,A -85,B 0,C 180,E1 -437.493,E2 -437.493} C_VEL
LIN {X 0,Y 608.487,Z 655.207,A -85,B 0,C 180,E1 -438.676,E2 -438.676} C_VEL
LIN {X 0,Y 608.471,Z 664.258,A -85,B 0,C 180,E1 -440.023,E2 -440.023} C_VEL
LIN {X 0,Y 608.444,Z 671.858,A -85,B 0,C 180,E1 -441.364,E2 -441.364} C_VEL
LIN {X 0,Y 608.437,Z 679.469,A -85,B 0,C 180,E1 -443.034,E2 -443.034} C_VEL
LIN {X 0,Y 608.435,Z 685.245,A -85,B 0,C 180,E1 -444.698,E2 -444.698} C_VEL
LIN {X 0,Y 608.431,Z 688.633,A -85,B 0,C 180,E1 -446.026,E2 -446.026} C_VEL
LIN {X 0,Y 608.412,Z 691.086,A -85,B 0,C 180,E1 -447.352,E2 -447.352} C_VEL
LIN {X 0,Y 608.441,Z 692.477,A -85,B 0,C 180,E1 -448.676,E2 -448.676} C_VEL
LIN {X 0,Y 608.429,Z 693,A -85,B 0,C 180,E1 -450,E2 -450} C_VEL
LIN {X 0,Y 608.441,Z 692.477,A -85,B 0,C 180,E1 -451.324,E2 -451.324} C_VEL
LIN {X 0,Y 608.412,Z 691.086,A -85,B 0,C 180,E1 -452.648,E2 -452.648} C_VEL
LIN {X 0,Y 608.431,Z 688.632,A -85,B 0,C 180,E1 -453.974,E2 -453.974} C_VEL
LIN {X 0,Y 608.435,Z 685.245,A -85,B 0,C 180,E1 -455.302,E2 -455.302} C_VEL
LIN {X 0,Y 608.437,Z 679.468,A -85,B 0,C 180,E1 -456.966,E2 -456.966} C_VEL
LIN {X 0,Y 608.444,Z 671.857,A -85,B 0,C 180,E1 -458.636,E2 -458.636} C_VEL
LIN {X 0,Y 608.462,Z 663.244,A -85,B 0,C 180,E1 -460.145,E2 -460.145} C_VEL
LIN {X 0,Y 608.466,Z 653.967,A -85,B 0,C 180,E1 -461.493,E2 -461.493} C_VEL
LIN {X 0,Y 608.49,Z 644.421,A -85,B 0,C 180,E1 -462.677,E2 -462.677} C_VEL
LIN {X 0,Y 608.521,Z 632.964,A -85,B 0,C 180,E1 -463.896,E2 -463.896} C_VEL
LIN {X 0,Y 608.553,Z 621.141,A -85,B 0,C 180,E1 -464.975,E2 -464.975} C_VEL
LIN {X 0,Y 608.607,Z 606.708,A -85,B 0,C 180,E1 -466.09,E2 -466.09} C_VEL
LIN {X 0,Y 608.623,Z 592.015,A -85,B 0,C 180,E1 -467.039,E2 -467.039} C_VEL
LIN {X 0,Y 608.659,Z 577.51,A -85,B 0,C 180,E1 -467.818,E2 -467.818} C_VEL
LIN {X 0,Y 608.718,Z 562.247,A -85,B 0,C 180,E1 -468.493,E2 -468.493} C_VEL
LIN {X 0,Y 608.748,Z 546.235,A -85,B 0,C 180,E1 -469.057,E2 -469.057} C_VEL
LIN {X 0,Y 608.787,Z 529.599,A -85,B 0,C 180,E1 -469.494,E2 -469.494} C_VEL
LIN {X 0,Y 608.807,Z 513.412,A -85,B 0,C 180,E1 -469.778,E2 -469.778} C_VEL
LIN {X 0,Y 608.918,Z 313.6,A -85,B 0,C 180,E1 -472.254,E2 -472.254} C_VEL
LIN {X 0,Y 608.726,Z 311.734,A -85,B 0,C 180,E1 -472.306,E2 -472.306} C_VEL
LIN {X 0,Y 608.774,Z 278.609,A -85,B 0,C 180,E1 -475.013,E2 -475.013} C_VEL
LIN {X 0,Y 608.827,Z 260.942,A -85,B 0,C 180,E1 -476.479,E2 -476.479} C_VEL
LIN {X 0,Y 608.432,Z 259.007,A -85,B 0,C 180,E1 -476.683,E2 -476.683} C_VEL
LIN {X 0,Y 608.433,Z 259.009,A -85,B 0,C 180,E1 -479.022,E2 -479.022} C_VEL
LIN {X 0,Y 608.459,Z 259.009,A -85,B 0,C 180,E1 -481.317,E2 -481.317} C_VEL
LIN {X 0,Y 608.475,Z 259,A -85,B 0,C 180,E1 -483.736,E2 -483.736} C_VEL
LIN {X 0,Y 608.445,Z 259.001,A -85,B 0,C 180,E1 -486.093,E2 -486.093} C_VEL
LIN {X 0,Y 608.464,Z 259,A -85,B 0,C 180,E1 -488.589,E2 -488.589} C_VEL
LIN {X 0,Y 608.46,Z 259.006,A -85,B 0,C 180,E1 -491.342,E2 -491.342} C_VEL
LIN {X 0,Y 608.457,Z 259,A -85,B 0,C 180,E1 -494.264,E2 -494.264} C_VEL
LIN {X 0,Y 608.456,Z 259.01,A -85,B 0,C 180,E1 -497.041,E2 -497.041} C_VEL
LIN {X 0,Y 608.452,Z 259.001,A -85,B 0,C 180,E1 -499.697,E2 -499.697} C_VEL
LIN {X 0,Y 608.467,Z 258.999,A -85,B 0,C 180,E1 -502.254,E2 -502.254} C_VEL
LIN {X 0,Y 608.447,Z 259.009,A -85,B 0,C 180,E1 -505.095,E2 -505.095} C_VEL
LIN {X 0,Y 608.459,Z 258.999,A -85,B 0,C 180,E1 -507.906,E2 -507.906} C_VEL
LIN {X 0,Y 608.472,Z 258.999,A -85,B 0,C 180,E1 -510.221,E2 -510.221} C_VEL
LIN {X 0,Y 608.444,Z 259.005,A -85,B 0,C 180,E1 -513.226,E2 -513.226} C_VEL
LIN {X 0,Y 608.481,Z 258.996,A -85,B 0,C 180,E1 -515.847,E2 -515.847} C_VEL
LIN {X 0,Y 608.471,Z 259,A -85,B 0,C 180,E1 -518.309,E2 -518.309} C_VEL
LIN {X 0,Y 608.458,Z 259.001,A -85,B 0,C 180,E1 -521.288,E2 -521.288} C_VEL
LIN {X 0,Y 608.456,Z 259,A -85,B 0,C 180,E1 -523.906,E2 -523.906} C_VEL
LIN {X 0,Y 608.464,Z 259.009,A -85,B 0,C 180,E1 -526.644,E2 -526.644} C_VEL
LIN {X 0,Y 608.439,Z 259.002,A -85,B 0,C 180,E1 -529.35,E2 -529.35} C_VEL
LIN {X 0,Y 608.48,Z 258.999,A -85,B 0,C 180,E1 -532.033,E2 -532.033} C_VEL
LIN {X 0,Y 608.457,Z 259.007,A -85,B 0,C 180,E1 -534.698,E2 -534.698} C_VEL
LIN {X 0,Y 608.446,Z 259.001,A -85,B 0,C 180,E1 -537.352,E2 -537.352} C_VEL
LIN {X 0,Y 608.477,Z 259,A -85,B 0,C 180,E1 -540,E2 -540} C_VEL
LIN {X 0,Y 608.467,Z 259.005,A -85,B 0,C 180,E1 -542.648,E2 -542.648} C_VEL
LIN {X 0,Y 608.427,Z 259.003,A -85,B 0,C 180,E1 -545.303,E2 -545.303} C_VEL
LIN {X 0,Y 608.473,Z 259.001,A -85,B 0,C 180,E1 -547.967,E2 -547.967} C_VEL
LIN {X 0,Y 608.428,Z 259.003,A -85,B 0,C 180,E1 -549.446,E2 -549.446} C_VEL
LIN {X 0,Y 607.769,Z 259.091,A -85,B 0,C 180,E1 -549.999,E2 -549.999} C_VEL
LIN {X 0,Y 604.93,Z 259.447,A -85,B 0,C 180,E1 -550.896,E2 -550.896} C_VEL
LIN {X 0,Y 602.525,Z 259.748,A -85,B 0,C 180,E1 -551.617,E2 -551.617} C_VEL
LIN {X 0,Y 601.484,Z 259.877,A -85,B 0,C 180,E1 -552.174,E2 -552.174} C_VEL
LIN {X 0,Y 601.395,Z 259.884,A -85,B 0,C 180,E1 -552.363,E2 -552.363} C_VEL
LIN {X 0,Y 601.384,Z 259.882,A -85,B 0,C 180,E1 -554.898,E2 -554.898} C_VEL
LIN {X 0,Y 601.373,Z 259.882,A -85,B 0,C 180,E1 -556.988,E2 -556.988} C_VEL
LIN {X 0,Y 601.384,Z 259.884,A -85,B 0,C 180,E1 -559.811,E2 -559.811} C_VEL
LIN {X 0,Y 601.379,Z 259.883,A -85,B 0,C 180,E1 -562.685,E2 -562.685} C_VEL
LIN {X 0,Y 601.367,Z 259.883,A -85,B 0,C 180,E1 -564.881,E2 -564.881} C_VEL
LIN {X 0,Y 601.363,Z 259.884,A -85,B 0,C 180,E1 -567.352,E2 -567.352} C_VEL
LIN {X 0,Y 601.405,Z 259.887,A -85,B 0,C 180,E1 -570.166,E2 -570.166} C_VEL
LIN {X 0,Y 601.382,Z 259.882,A -85,B 0,C 180,E1 -572.709,E2 -572.709} C_VEL
LIN {X 0,Y 601.344,Z 259.885,A -85,B 0,C 180,E1 -575.105,E2 -575.105} C_VEL
LIN {X 0,Y 601.382,Z 259.884,A -85,B 0,C 180,E1 -577.423,E2 -577.423} C_VEL
LIN {X 0,Y 601.378,Z 259.89,A -85,B 0,C 180,E1 -579.998,E2 -579.998} C_VEL
LIN {X 0,Y 601.353,Z 259.885,A -85,B 0,C 180,E1 -582.676,E2 -582.676} C_VEL
LIN {X 0,Y 601.403,Z 259.883,A -85,B 0,C 180,E1 -585.48,E2 -585.48} C_VEL
LIN {X 0,Y 601.403,Z 259.88,A -85,B 0,C 180,E1 -588.41,E2 -588.41} C_VEL
LIN {X 0,Y 601.378,Z 259.883,A -85,B 0,C 180,E1 -590.871,E2 -590.871} C_VEL
LIN {X 0,Y 601.438,Z 260.051,A -85,B 0,C 180,E1 -592.344,E2 -592.344} C_VEL
LIN {X 0,Y 601.914,Z 263.637,A -85,B 0,C 180,E1 -592.704,E2 -592.704} C_VEL
LIN {X 0,Y 601.879,Z 283.079,A -85,B 0,C 180,E1 -594.51,E2 -594.51} C_VEL
LIN {X 0,Y 602.312,Z 286.957,A -85,B 0,C 180,E1 -594.576,E2 -594.576} C_VEL
LIN {X 0,Y 602.132,Z 488.935,A -85,B 0,C 180,E1 -597.12,E2 -597.12} C_VEL
LIN {X 0,Y 602.072,Z 504.899,A -85,B 0,C 180,E1 -597.454,E2 -597.454} C_VEL
LIN {X 0,Y 601.998,Z 520.738,A -85,B 0,C 180,E1 -597.914,E2 -597.914} C_VEL
LIN {X 0,Y 601.912,Z 536.563,A -85,B 0,C 180,E1 -598.512,E2 -598.512} C_VEL
LIN {X 0,Y 601.849,Z 550.716,A -85,B 0,C 180,E1 -599.18,E2 -599.18} C_VEL
LIN {X 0,Y 601.77,Z 564.358,A -85,B 0,C 180,E1 -599.951,E2 -599.951} C_VEL
LIN {X 0,Y 601.694,Z 578.036,A -85,B 0,C 180,E1 -600.864,E2 -600.864} C_VEL
LIN {X 0,Y 601.615,Z 591.825,A -85,B 0,C 180,E1 -601.953,E2 -601.953} C_VEL
LIN {X 0,Y 601.549,Z 603.964,A -85,B 0,C 180,E1 -603.081,E2 -603.081} C_VEL
LIN {X 0,Y 601.474,Z 614.231,A -85,B 0,C 180,E1 -604.196,E2 -604.196} C_VEL
LIN {X 0,Y 601.425,Z 624.228,A -85,B 0,C 180,E1 -605.452,E2 -605.452} C_VEL
LIN {X 0,Y 601.4,Z 633.197,A -85,B 0,C 180,E1 -606.771,E2 -606.771} C_VEL
LIN {X 0,Y 601.374,Z 640.43,A -85,B 0,C 180,E1 -608.039,E2 -608.039} C_VEL
LIN {X 0,Y 601.353,Z 647.275,A -85,B 0,C 180,E1 -609.475,E2 -609.475} C_VEL
LIN {X 0,Y 601.334,Z 652.778,A -85,B 0,C 180,E1 -610.898,E2 -610.898} C_VEL
LIN {X 0,Y 601.31,Z 656.942,A -85,B 0,C 180,E1 -612.309,E2 -612.309} C_VEL
LIN {X 0,Y 601.342,Z 660.008,A -85,B 0,C 180,E1 -613.71,E2 -613.71} C_VEL
LIN {X 0,Y 601.313,Z 661.964,A -85,B 0,C 180,E1 -615.1,E2 -615.1} C_VEL
LIN {X 0,Y 601.336,Z 662.875,A -85,B 0,C 180,E1 -616.482,E2 -616.482} C_VEL
LIN {X 0,Y 601.338,Z 662.817,A -85,B 0,C 180,E1 -617.856,E2 -617.856} C_VEL
LIN {X 0,Y 601.329,Z 661.693,A -85,B 0,C 180,E1 -619.222,E2 -619.222} C_VEL
LIN {X 0,Y 601.334,Z 659.663,A -85,B 0,C 180,E1 -620.583,E2 -620.583} C_VEL
LIN {X 0,Y 601.331,Z 656.528,A -85,B 0,C 180,E1 -621.938,E2 -621.938} C_VEL
LIN {X 0,Y 601.354,Z 651.979,A -85,B 0,C 180,E1 -623.413,E2 -623.413} C_VEL
LIN {X 0,Y 601.36,Z 645.75,A -85,B 0,C 180,E1 -624.971,E2 -624.971} C_VEL
LIN {X 0,Y 601.362,Z 639.018,A -85,B 0,C 180,E1 -626.315,E2 -626.315} C_VEL
LIN {X 0,Y 601.416,Z 631.018,A -85,B 0,C 180,E1 -627.656,E2 -627.656} C_VEL
LIN {X 0,Y 601.45,Z 621.572,A -85,B 0,C 180,E1 -628.996,E2 -628.996} C_VEL
LIN {X 0,Y 601.513,Z 610.38,A -85,B 0,C 180,E1 -630.335,E2 -630.335} C_VEL
LIN {X 0,Y 601.554,Z 598.84,A -85,B 0,C 180,E1 -631.506,E2 -631.506} C_VEL
LIN {X 0,Y 601.635,Z 586.292,A -85,B 0,C 180,E1 -632.594,E2 -632.594} C_VEL
LIN {X 0,Y 601.69,Z 572.707,A -85,B 0,C 180,E1 -633.599,E2 -633.599} C_VEL
LIN {X 0,Y 601.787,Z 557.885,A -85,B 0,C 180,E1 -634.521,E2 -634.521} C_VEL
LIN {X 0,Y 601.88,Z 543.342,A -85,B 0,C 180,E1 -635.276,E2 -635.276} C_VEL
LIN {X 0,Y 601.994,Z 527.294,A -85,B 0,C 180,E1 -635.947,E2 -635.947} C_VEL
LIN {X 0,Y 602.059,Z 511.392,A -85,B 0,C 180,E1 -636.464,E2 -636.464} C_VEL
LIN {X 0,Y 602.107,Z 494.888,A -85,B 0,C 180,E1 -636.859,E2 -636.859} C_VEL
LIN {X 0,Y 602.135,Z 478.597,A -85,B 0,C 180,E1 -637.118,E2 -637.118} C_VEL
LIN {X 0,Y 602.322,Z 285.777,A -85,B 0,C 180,E1 -639.529,E2 -639.529} C_VEL
LIN {X 0,Y 601.869,Z 282.716,A -85,B 0,C 180,E1 -639.6,E2 -639.6} C_VEL
LIN {X 0,Y 601.952,Z 262.965,A -85,B 0,C 180,E1 -641.448,E2 -641.448} C_VEL
LIN {X 0,Y 601.406,Z 259.884,A -85,B 0,C 180,E1 -641.779,E2 -641.779} C_VEL
LIN {X 0,Y 601.418,Z 259.886,A -85,B 0,C 180,E1 -644.205,E2 -644.205} C_VEL
LIN {X 0,Y 601.377,Z 259.882,A -85,B 0,C 180,E1 -646.987,E2 -646.987} C_VEL
LIN {X 0,Y 601.387,Z 259.884,A -85,B 0,C 180,E1 -649.81,E2 -649.81} C_VEL
LIN {X 0,Y 601.4,Z 259.882,A -85,B 0,C 180,E1 -652.683,E2 -652.683} C_VEL
LIN {X 0,Y 601.372,Z 259.883,A -85,B 0,C 180,E1 -654.88,E2 -654.88} C_VEL
LIN {X 0,Y 601.368,Z 259.883,A -85,B 0,C 180,E1 -657.352,E2 -657.352} C_VEL
LIN {X 0,Y 601.407,Z 259.888,A -85,B 0,C 180,E1 -660.165,E2 -660.165} C_VEL
LIN {X 0,Y 601.39,Z 259.881,A -85,B 0,C 180,E1 -662.71,E2 -662.71} C_VEL
LIN {X 0,Y 601.347,Z 259.885,A -85,B 0,C 180,E1 -665.104,E2 -665.104} C_VEL
LIN {X 0,Y 601.364,Z 259.884,A -85,B 0,C 180,E1 -667.424,E2 -667.424} C_VEL
LIN {X 0,Y 601.376,Z 259.892,A -85,B 0,C 180,E1 -669.998,E2 -669.998} C_VEL
LIN {X 0,Y 601.346,Z 259.886,A -85,B 0,C 180,E1 -672.676,E2 -672.676} C_VEL
LIN {X 0,Y 601.367,Z 259.885,A -85,B 0,C 180,E1 -674.529,E2 -674.529} C_VEL
LIN {X 0,Y 601.402,Z 259.881,A -85,B 0,C 180,E1 -676.43,E2 -676.43} C_VEL
LIN {X 0,Y 601.351,Z 259.885,A -85,B 0,C 180,E1 -679.12,E2 -679.12} C_VEL
LIN {X 0,Y 601.409,Z 259.885,A -85,B 0,C 180,E1 -681.731,E2 -681.731} C_VEL
LIN {X 0,Y 601.374,Z 259.884,A -85,B 0,C 180,E1 -684.244,E2 -684.244} C_VEL
LIN {X 0,Y 601.383,Z 259.88,A -85,B 0,C 180,E1 -686.683,E2 -686.683} C_VEL
LIN {X 0,Y 601.389,Z 259.881,A -85,B 0,C 180,E1 -689.056,E2 -689.056} C_VEL
LIN {X 0,Y 601.381,Z 259.884,A -85,B 0,C 180,E1 -691.37,E2 -691.37} C_VEL
LIN {X 0,Y 601.391,Z 259.881,A -85,B 0,C 180,E1 -694.38,E2 -694.38} C_VEL
LIN {X 0,Y 601.376,Z 259.881,A -85,B 0,C 180,E1 -696.587,E2 -696.587} C_VEL
LIN {X 0,Y 601.421,Z 259.883,A -85,B 0,C 180,E1 -699.477,E2 -699.477} C_VEL
LIN {X 0,Y 601.379,Z 259.882,A -85,B 0,C 180,E1 -702.311,E2 -702.311} C_VEL
LIN {X 0,Y 601.393,Z 259.88,A -85,B 0,C 180,E1 -704.408,E2 -704.408} C_VEL
LIN {X 0,Y 601.403,Z 259.882,A -85,B 0,C 180,E1 -707.171,E2 -707.171} C_VEL
LIN {X 0,Y 601.43,Z 259.879,A -85,B 0,C 180,E1 -709.905,E2 -709.905} C_VEL
LIN {X 0,Y 601.379,Z 259.881,A -85,B 0,C 180,E1 -712.614,E2 -712.614} C_VEL
LIN {X 0,Y 601.423,Z 259.883,A -85,B 0,C 180,E1 -715.308,E2 -715.308} C_VEL
LIN {X 0,Y 601.435,Z 259.876,A -85,B 0,C 180,E1 -717.991,E2 -717.991} C_VEL
LIN {X 0,Y 601.427,Z 259.875,A -85,B 0,C 180,E1 -720.669,E2 -720.669} C_VEL
LIN {X 0,Y 601.428,Z 259.885,A -85,B 0,C 180,E1 -723.349,E2 -723.349} C_VEL
LIN {X 0,Y 601.432,Z 259.875,A -85,B 0,C 180,E1 -726.037,E2 -726.037} C_VEL
LIN {X 0,Y 601.403,Z 259.879,A -85,B 0,C 180,E1 -728.738,E2 -728.738} C_VEL
LIN {X 0,Y 601.437,Z 259.881,A -85,B 0,C 180,E1 -731.458,E2 -731.458} C_VEL
LIN {X 0,Y 601.416,Z 259.876,A -85,B 0,C 180,E1 -734.205,E2 -734.205} C_VEL
LIN {X 0,Y 601.414,Z 259.883,A -85,B 0,C 180,E1 -736.986,E2 -736.986} C_VEL
LIN {X 0,Y 601.406,Z 259.879,A -85,B 0,C 180,E1 -739.809,E2 -739.809} C_VEL
LIN {X 0,Y 601.412,Z 259.88,A -85,B 0,C 180,E1 -742.683,E2 -742.683} C_VEL
LIN {X 0,Y 601.401,Z 259.885,A -85,B 0,C 180,E1 -744.878,E2 -744.878} C_VEL
LIN {X 0,Y 601.42,Z 259.882,A -85,B 0,C 180,E1 -747.363,E2 -747.363} C_VEL
LIN {X 0,Y 601.428,Z 259.875,A -85,B 0,C 180,E1 -750.164,E2 -750.164} C_VEL
LIN {X 0,Y 601.415,Z 259.882,A -85,B 0,C 180,E1 -752.714,E2 -752.714} C_VEL
LIN {X 0,Y 601.396,Z 259.887,A -85,B 0,C 180,E1 -755.112,E2 -755.112} C_VEL
LIN {X 0,Y 601.434,Z 259.877,A -85,B 0,C 180,E1 -757.419,E2 -757.419} C_VEL
LIN {X 0,Y 601.411,Z 259.877,A -85,B 0,C 180,E1 -759.995,E2 -759.995} C_VEL
LIN {X 0,Y 601.411,Z 259.884,A -85,B 0,C 180,E1 -762.67,E2 -762.67} C_VEL
LIN {X 0,Y 601.425,Z 259.877,A -85,B 0,C 180,E1 -765.482,E2 -765.482} C_VEL
LIN {X 0,Y 601.424,Z 259.879,A -85,B 0,C 180,E1 -768.406,E2 -768.406} C_VEL
LIN {X 0,Y 601.434,Z 259.884,A -85,B 0,C 180,E1 -770.875,E2 -770.875} C_VEL
LIN {X 0,Y 601.405,Z 259.878,A -85,B 0,C 180,E1 -773.739,E2 -773.739} C_VEL
LIN {X 0,Y 601.425,Z 259.885,A -85,B 0,C 180,E1 -776.686,E2 -776.686} C_VEL
LIN {X 0,Y 601.417,Z 259.882,A -85,B 0,C 180,E1 -779.058,E2 -779.058} C_VEL
LIN {X 0,Y 601.412,Z 259.88,A -85,B 0,C 180,E1 -781.372,E2 -781.372} C_VEL
LIN {X 0,Y 601.433,Z 259.978,A -85,B 0,C 180,E1 -783.088,E2 -783.088} C_VEL
LIN {X 0,Y 602.18,Z 263.153,A -85,B 0,C 180,E1 -783.393,E2 -783.393} C_VEL
LIN {X 0,Y 602.013,Z 295.174,A -85,B 0,C 180,E1 -786.066,E2 -786.066} C_VEL
LIN {X 0,Y 601.96,Z 312.018,A -85,B 0,C 180,E1 -787.453,E2 -787.453} C_VEL
LIN {X 0,Y 602.356,Z 315.845,A -85,B 0,C 180,E1 -787.519,E2 -787.519} C_VEL
LIN {X 0,Y 602.124,Z 517.941,A -85,B 0,C 180,E1 -790.06,E2 -790.06} C_VEL
LIN {X 0,Y 602.075,Z 534.175,A -85,B 0,C 180,E1 -790.391,E2 -790.391} C_VEL
LIN {X 0,Y 602.011,Z 550.94,A -85,B 0,C 180,E1 -790.876,E2 -790.876} C_VEL
LIN {X 0,Y 601.915,Z 566.239,A -85,B 0,C 180,E1 -791.452,E2 -791.452} C_VEL
LIN {X 0,Y 601.868,Z 581.013,A -85,B 0,C 180,E1 -792.15,E2 -792.15} C_VEL
LIN {X 0,Y 601.767,Z 594.843,A -85,B 0,C 180,E1 -792.936,E2 -792.936} C_VEL
LIN {X 0,Y 601.696,Z 609.049,A -85,B 0,C 180,E1 -793.895,E2 -793.895} C_VEL
LIN {X 0,Y 601.592,Z 622.127,A -85,B 0,C 180,E1 -794.934,E2 -794.934} C_VEL
LIN {X 0,Y 601.555,Z 634.678,A -85,B 0,C 180,E1 -796.108,E2 -796.108} C_VEL
LIN {X 0,Y 601.472,Z 645.911,A -85,B 0,C 180,E1 -797.345,E2 -797.345} C_VEL
LIN {X 0,Y 601.427,Z 656.287,A -85,B 0,C 180,E1 -798.691,E2 -798.691} C_VEL
LIN {X 0,Y 601.387,Z 665.272,A -85,B 0,C 180,E1 -800.074,E2 -800.074} C_VEL
LIN {X 0,Y 601.365,Z 673.486,A -85,B 0,C 180,E1 -801.6,E2 -801.6} C_VEL
LIN {X 0,Y 601.361,Z 679.468,A -85,B 0,C 180,E1 -802.951,E2 -802.951} C_VEL
LIN {X 0,Y 601.345,Z 685.246,A -85,B 0,C 180,E1 -804.635,E2 -804.635} C_VEL
LIN {X 0,Y 601.34,Z 688.633,A -85,B 0,C 180,E1 -805.979,E2 -805.979} C_VEL
LIN {X 0,Y 601.311,Z 691.086,A -85,B 0,C 180,E1 -807.32,E2 -807.32} C_VEL
LIN {X 0,Y 601.34,Z 692.477,A -85,B 0,C 180,E1 -808.661,E2 -808.661} C_VEL
LIN {X 0,Y 601.33,Z 693,A -85,B 0,C 180,E1 -810,E2 -810} C_VEL
LIN {X 0,Y 601.34,Z 692.477,A -85,B 0,C 180,E1 -811.339,E2 -811.339} C_VEL
LIN {X 0,Y 601.311,Z 691.086,A -85,B 0,C 180,E1 -812.68,E2 -812.68} C_VEL
LIN {X 0,Y 601.34,Z 688.633,A -85,B 0,C 180,E1 -814.021,E2 -814.021} C_VEL
LIN {X 0,Y 601.345,Z 685.246,A -85,B 0,C 180,E1 -815.365,E2 -815.365} C_VEL
LIN {X 0,Y 601.362,Z 679.468,A -85,B 0,C 180,E1 -817.049,E2 -817.049} C_VEL
LIN {X 0,Y 601.376,Z 671.857,A -85,B 0,C 180,E1 -818.739,E2 -818.739} C_VEL
LIN {X 0,Y 601.411,Z 663.246,A -85,B 0,C 180,E1 -820.266,E2 -820.266} C_VEL
LIN {X 0,Y 601.429,Z 653.968,A -85,B 0,C 180,E1 -821.629,E2 -821.629} C_VEL
LIN {X 0,Y 601.479,Z 644.421,A -85,B 0,C 180,E1 -822.827,E2 -822.827} C_VEL
LIN {X 0,Y 601.544,Z 633.618,A -85,B 0,C 180,E1 -823.997,E2 -823.997} C_VEL
LIN {X 0,Y 601.606,Z 621.142,A -85,B 0,C 180,E1 -825.152,E2 -825.152} C_VEL
LIN {X 0,Y 601.707,Z 607.883,A -85,B 0,C 180,E1 -826.192,E2 -826.192} C_VEL
LIN {X 0,Y 601.764,Z 593.429,A -85,B 0,C 180,E1 -827.151,E2 -827.151} C_VEL
LIN {X 0,Y 601.863,Z 579.261,A -85,B 0,C 180,E1 -827.938,E2 -827.938} C_VEL
LIN {X 0,Y 601.942,Z 564.909,A -85,B 0,C 180,E1 -828.604,E2 -828.604} C_VEL
LIN {X 0,Y 602.011,Z 548.343,A -85,B 0,C 180,E1 -829.212,E2 -829.212} C_VEL
LIN {X 0,Y 602.09,Z 532.344,A -85,B 0,C 180,E1 -829.653,E2 -829.653} C_VEL
LIN {X 0,Y 602.142,Z 516.425,A -85,B 0,C 180,E1 -829.962,E2 -829.962} C_VEL
LIN {X 0,Y 602.322,Z 314.072,A -85,B 0,C 180,E1 -832.505,E2 -832.505} C_VEL
LIN {X 0,Y 601.968,Z 311.813,A -85,B 0,C 180,E1 -832.564,E2 -832.564} C_VEL
LIN {X 0,Y 602.109,Z 277.505,A -85,B 0,C 180,E1 -835.402,E2 -835.402} C_VEL
LIN {X 0,Y 602.18,Z 263.151,A -85,B 0,C 180,E1 -836.607,E2 -836.607} C_VEL
LIN {X 0,Y 601.408,Z 259.886,A -85,B 0,C 180,E1 -836.925,E2 -836.925} C_VEL
LIN {X 0,Y 601.406,Z 259.888,A -85,B 0,C 180,E1 -839.394,E2 -839.394} C_VEL
LIN {X 0,Y 601.404,Z 259.882,A -85,B 0,C 180,E1 -841.727,E2 -841.727} C_VEL
LIN {X 0,Y 601.426,Z 259.876,A -85,B 0,C 180,E1 -844.119,E2 -844.119} C_VEL
LIN {X 0,Y 601.436,Z 259.882,A -85,B 0,C 180,E1 -847.383,E2 -847.383} C_VEL
LIN {X 0,Y 601.41,Z 259.878,A -85,B 0,C 180,E1 -849.995,E2 -849.995} C_VEL
LIN {X 0,Y 601.409,Z 259.88,A -85,B 0,C 180,E1 -852.671,E2 -852.671} C_VEL
LIN {X 0,Y 601.426,Z 259.879,A -85,B 0,C 180,E1 -855.482,E2 -855.482} C_VEL
LIN {X 0,Y 601.424,Z 259.877,A -85,B 0,C 180,E1 -858.407,E2 -858.407} C_VEL
LIN {X 0,Y 601.437,Z 259.882,A -85,B 0,C 180,E1 -860.876,E2 -860.876} C_VEL
LIN {X 0,Y 601.405,Z 259.881,A -85,B 0,C 180,E1 -863.418,E2 -863.418} C_VEL
LIN {X 0,Y 601.432,Z 259.874,A -85,B 0,C 180,E1 -866.065,E2 -866.065} C_VEL
LIN {X 0,Y 601.43,Z 259.879,A -85,B 0,C 180,E1 -868.544,E2 -868.544} C_VEL
LIN {X 0,Y 601.421,Z 259.877,A -85,B 0,C 180,E1 -871.373,E2 -871.373} C_VEL
LIN {X 0,Y 601.398,Z 259.879,A -85,B 0,C 180,E1 -873.636,E2 -873.636} C_VEL
LIN {X 0,Y 601.418,Z 259.883,A -85,B 0,C 180,E1 -876.59,E2 -876.59} C_VEL
LIN {X 0,Y 601.418,Z 259.877,A -85,B 0,C 180,E1 -879.478,E2 -879.478} C_VEL
LIN {X 0,Y 601.402,Z 259.882,A -85,B 0,C 180,E1 -882.312,E2 -882.312} C_VEL
LIN {X 0,Y 601.413,Z 259.882,A -85,B 0,C 180,E1 -884.409,E2 -884.409} C_VEL
LIN {X 0,Y 601.405,Z 259.88,A -85,B 0,C 180,E1 -887.172,E2 -887.172} C_VEL
LIN {X 0,Y 601.43,Z 259.875,A -85,B 0,C 180,E1 -889.905,E2 -889.905} C_VEL
LIN {X 0,Y 601.41,Z 259.887,A -85,B 0,C 180,E1 -892.615,E2 -892.615} C_VEL
LIN {X 0,Y 601.395,Z 259.878,A -85,B 0,C 180,E1 -895.308,E2 -895.308} C_VEL
LIN {X 0,Y 601.434,Z 259.877,A -85,B 0,C 180,E1 -897.991,E2 -897.991} C_VEL
LIN {X 0,Y 601.442,Z 259.879,A -85,B 0,C 180,E1 -900.67,E2 -900.67} C_VEL
LIN {X 0,Y 601.37,Z 259.882,A -85,B 0,C 180,E1 -903.35,E2 -903.35} C_VEL
LIN {X 0,Y 601.408,Z 259.882,A -85,B 0,C 180,E1 -906.038,E2 -906.038} C_VEL
LIN {X 0,Y 601.398,Z 259.882,A -85,B 0,C 180,E1 -908.739,E2 -908.739} C_VEL
LIN {X 0,Y 601.4,Z 259.879,A -85,B 0,C 180,E1 -911.459,E2 -911.459} C_VEL
LIN {X 0,Y 601.395,Z 259.884,A -85,B 0,C 180,E1 -912.363,E2 -912.363} C_VEL
LIN {X 0,Y 600.716,Z 259.965,A -85,B 0,C 180,E1 -912.922,E2 -912.922} C_VEL
LIN {X 0,Y 597.856,Z 260.322,A -85,B 0,C 180,E1 -913.83,E2 -913.83} C_VEL
LIN {X 0,Y 595.446,Z 260.625,A -85,B 0,C 180,E1 -914.56,E2 -914.56} C_VEL
LIN {X 0,Y 594.412,Z 260.749,A -85,B 0,C 180,E1 -915.124,E2 -915.124} C_VEL
LIN {X 0,Y 594.328,Z 260.759,A -85,B 0,C 180,E1 -915.315,E2 -915.315} C_VEL
LIN {X 0,Y 594.329,Z 260.765,A -85,B 0,C 180,E1 -917.906,E2 -917.906} C_VEL
LIN {X 0,Y 594.381,Z 260.755,A -85,B 0,C 180,E1 -920.777,E2 -920.777} C_VEL
LIN {X 0,Y 594.354,Z 260.759,A -85,B 0,C 180,E1 -923.706,E2 -923.706} C_VEL
LIN {X 0,Y 594.333,Z 260.76,A -85,B 0,C 180,E1 -926.703,E2 -926.703} C_VEL
LIN {X 0,Y 594.35,Z 260.762,A -85,B 0,C 180,E1 -929.778,E2 -929.778} C_VEL
LIN {X 0,Y 594.335,Z 260.767,A -85,B 0,C 180,E1 -932.15,E2 -932.15} C_VEL
LIN {X 0,Y 594.323,Z 260.762,A -85,B 0,C 180,E1 -934.584,E2 -934.584} C_VEL
LIN {X 0,Y 594.316,Z 260.762,A -85,B 0,C 180,E1 -937.092,E2 -937.092} C_VEL
LIN {X 0,Y 594.335,Z 260.767,A -85,B 0,C 180,E1 -939.769,E2 -939.769} C_VEL
LIN {X 0,Y 594.329,Z 260.763,A -85,B 0,C 180,E1 -942.38,E2 -942.38} C_VEL
LIN {X 0,Y 594.332,Z 260.761,A -85,B 0,C 180,E1 -945.195,E2 -945.195} C_VEL
LIN {X 0,Y 594.375,Z 260.759,A -85,B 0,C 180,E1 -948.153,E2 -948.153} C_VEL
LIN {X 0,Y 594.365,Z 260.76,A -85,B 0,C 180,E1 -951.299,E2 -951.299} C_VEL
LIN {X 0,Y 594.408,Z 260.862,A -85,B 0,C 180,E1 -952.11,E2 -952.11} C_VEL
LIN {X 0,Y 595.163,Z 265.519,A -85,B 0,C 180,E1 -952.589,E2 -952.589} C_VEL
LIN {X 0,Y 595.138,Z 283.236,A -85,B 0,C 180,E1 -954.242,E2 -954.242} C_VEL
LIN {X 0,Y 595.754,Z 287.275,A -85,B 0,C 180,E1 -954.319,E2 -954.319} C_VEL
LIN {X 0,Y 595.457,Z 489.251,A -85,B 0,C 180,E1 -956.891,E2 -956.891} C_VEL
LIN {X 0,Y 595.377,Z 505.963,A -85,B 0,C 180,E1 -957.25,E2 -957.25} C_VEL
LIN {X 0,Y 595.264,Z 521.261,A -85,B 0,C 180,E1 -957.707,E2 -957.707} C_VEL
LIN {X 0,Y 595.135,Z 536.946,A -85,B 0,C 180,E1 -958.31,E2 -958.31} C_VEL
LIN {X 0,Y 595.031,Z 551.048,A -85,B 0,C 180,E1 -958.985,E2 -958.985} C_VEL
LIN {X 0,Y 594.915,Z 565.014,A -85,B 0,C 180,E1 -959.789,E2 -959.789} C_VEL
LIN {X 0,Y 594.774,Z 578.984,A -85,B 0,C 180,E1 -960.742,E2 -960.742} C_VEL
LIN {X 0,Y 594.663,Z 591.996,A -85,B 0,C 180,E1 -961.788,E2 -961.788} C_VEL
LIN {X 0,Y 594.556,Z 604.118,A -85,B 0,C 180,E1 -962.929,E2 -962.929} C_VEL
LIN {X 0,Y 594.456,Z 615.996,A -85,B 0,C 180,E1 -964.248,E2 -964.248} C_VEL
LIN {X 0,Y 594.405,Z 626.029,A -85,B 0,C 180,E1 -965.564,E2 -965.564} C_VEL
LIN {X 0,Y 594.357,Z 634.376,A -85,B 0,C 180,E1 -966.848,E2 -966.848} C_VEL
LIN {X 0,Y 594.302,Z 641.48,A -85,B 0,C 180,E1 -968.13,E2 -968.13} C_VEL
LIN {X 0,Y 594.282,Z 648.097,A -85,B 0,C 180,E1 -969.582,E2 -969.582} C_VEL
LIN {X 0,Y 594.243,Z 653.676,A -85,B 0,C 180,E1 -971.112,E2 -971.112} C_VEL
LIN {X 0,Y 594.209,Z 656.52,A -85,B 0,C 180,E1 -972.09,E2 -972.09} C_VEL
LIN {X 0,Y 594.238,Z 659.744,A -85,B 0,C 180,E1 -973.51,E2 -973.51} C_VEL
LIN {X 0,Y 594.208,Z 661.782,A -85,B 0,C 180,E1 -974.918,E2 -974.918} C_VEL
LIN {X 0,Y 594.255,Z 662.839,A -85,B 0,C 180,E1 -976.318,E2 -976.318} C_VEL
LIN {X 0,Y 594.235,Z 662.853,A -85,B 0,C 180,E1 -977.708,E2 -977.708} C_VEL
LIN {X 0,Y 594.243,Z 661.874,A -85,B 0,C 180,E1 -979.092,E2 -979.092} C_VEL
LIN {X 0,Y 594.253,Z 659.927,A -85,B 0,C 180,E1 -980.469,E2 -980.469} C_VEL
LIN {X 0,Y 594.227,Z 656.935,A -85,B 0,C 180,E1 -981.841,E2 -981.841} C_VEL
LIN {X 0,Y 594.272,Z 652.233,A -85,B 0,C 180,E1 -983.42,E2 -983.42} C_VEL
LIN {X 0,Y 594.271,Z 646.417,A -85,B 0,C 180,E1 -984.911,E2 -984.911} C_VEL
LIN {X 0,Y 594.288,Z 639.841,A -85,B 0,C 180,E1 -986.271,E2 -986.271} C_VEL
LIN {X 0,Y 594.382,Z 630.924,A -85,B 0,C 180,E1 -987.798,E2 -987.798} C_VEL
LIN {X 0,Y 594.421,Z 621.461,A -85,B 0,C 180,E1 -989.153,E2 -989.153} C_VEL
LIN {X 0,Y 594.501,Z 610.253,A -85,B 0,C 180,E1 -990.508,E2 -990.508} C_VEL
LIN {X 0,Y 594.591,Z 598.697,A -85,B 0,C 180,E1 -991.693,E2 -991.693} C_VEL
LIN {X 0,Y 594.716,Z 586.125,A -85,B 0,C 180,E1 -992.794,E2 -992.794} C_VEL
LIN {X 0,Y 594.798,Z 572.509,A -85,B 0,C 180,E1 -993.811,E2 -993.811} C_VEL
LIN {X 0,Y 594.957,Z 557.632,A -85,B 0,C 180,E1 -994.743,E2 -994.743} C_VEL
LIN {X 0,Y 595.087,Z 543.019,A -85,B 0,C 180,E1 -995.506,E2 -995.506} C_VEL
LIN {X 0,Y 595.249,Z 526.992,A -85,B 0,C 180,E1 -996.181,E2 -996.181} C_VEL
LIN {X 0,Y 595.338,Z 511.421,A -85,B 0,C 180,E1 -996.691,E2 -996.691} C_VEL
LIN {X 0,Y 595.423,Z 495.283,A -85,B 0,C 180,E1 -997.083,E2 -997.083} C_VEL
LIN {X 0,Y 595.482,Z 477.99,A -85,B 0,C 180,E1 -997.36,E2 -997.36} C_VEL
LIN {X 0,Y 595.773,Z 287.856,A -85,B 0,C 180,E1 -999.763,E2 -999.763} C_VEL
LIN {X 0,Y 595.293,Z 283.929,A -85,B 0,C 180,E1 -999.833,E2 -999.833} C_VEL
LIN {X 0,Y 595.083,Z 282.832,A -85,B 0,C 180,E1 -999.86,E2 -999.86} C_VEL
LIN {X 0,Y 595.194,Z 264.676,A -85,B 0,C 180,E1 -1001.58,E2 -1001.58} C_VEL
LIN {X 0,Y 594.391,Z 260.761,A -85,B 0,C 180,E1 -1002.007,E2 -1002.007} C_VEL
LIN {X 0,Y 594.385,Z 260.763,A -85,B 0,C 180,E1 -1004.377,E2 -1004.377} C_VEL
LIN {X 0,Y 594.328,Z 260.76,A -85,B 0,C 180,E1 -1007.195,E2 -1007.195} C_VEL
LIN {X 0,Y 594.359,Z 260.763,A -85,B 0,C 180,E1 -1010.054,E2 -1010.054} C_VEL
LIN {X 0,Y 594.346,Z 260.758,A -85,B 0,C 180,E1 -1012.968,E2 -1012.968} C_VEL
LIN {X 0,Y 594.322,Z 260.76,A -85,B 0,C 180,E1 -1015.195,E2 -1015.195} C_VEL
LIN {X 0,Y 594.328,Z 260.761,A -85,B 0,C 180,E1 -1017.515,E2 -1017.515} C_VEL
LIN {X 0,Y 594.368,Z 260.762,A -85,B 0,C 180,E1 -1020.324,E2 -1020.324} C_VEL
LIN {X 0,Y 594.338,Z 260.759,A -85,B 0,C 180,E1 -1022.953,E2 -1022.953} C_VEL
LIN {X 0,Y 594.304,Z 260.763,A -85,B 0,C 180,E1 -1025.412,E2 -1025.412} C_VEL
LIN {X 0,Y 594.311,Z 260.771,A -85,B 0,C 180,E1 -1027.946,E2 -1027.946} C_VEL
LIN {X 0,Y 594.323,Z 260.762,A -85,B 0,C 180,E1 -1030.571,E2 -1030.571} C_VEL
LIN {X 0,Y 594.31,Z 260.762,A -85,B 0,C 180,E1 -1032.846,E2 -1032.846} C_VEL
LIN {X 0,Y 594.308,Z 260.762,A -85,B 0,C 180,E1 -1035.197,E2 -1035.197} C_VEL
LIN {X 0,Y 594.37,Z 260.761,A -85,B 0,C 180,E1 -1038.153,E2 -1038.153} C_VEL
LIN {X 0,Y 594.36,Z 260.757,A -85,B 0,C 180,E1 -1041.299,E2 -1041.299} C_VEL
LIN {X 0,Y 594.341,Z 260.764,A -85,B 0,C 180,E1 -1043.754,E2 -1043.754} C_VEL
LIN {X 0,Y 594.354,Z 260.76,A -85,B 0,C 180,E1 -1046.237,E2 -1046.237} C_VEL
LIN {X 0,Y 594.355,Z 260.756,A -85,B 0,C 180,E1 -1048.648,E2 -1048.648} C_VEL
LIN {X 0,Y 594.338,Z 260.758,A -85,B 0,C 180,E1 -1051.05,E2 -1051.05} C_VEL
LIN {X 0,Y 594.351,Z 260.762,A -85,B 0,C 180,E1 -1053.984,E2 -1053.984} C_VEL
LIN {X 0,Y 594.369,Z 260.755,A -85,B 0,C 180,E1 -1056.295,E2 -1056.295} C_VEL
LIN {X 0,Y 594.392,Z 260.755,A -85,B 0,C 180,E1 -1059.224,E2 -1059.224} C_VEL
LIN {X 0,Y 594.339,Z 260.76,A -85,B 0,C 180,E1 -1062.094,E2 -1062.094} C_VEL
LIN {X 0,Y 594.349,Z 260.758,A -85,B 0,C 180,E1 -1064.218,E2 -1064.218} C_VEL
LIN {X 0,Y 594.369,Z 260.755,A -85,B 0,C 180,E1 -1066.32,E2 -1066.32} C_VEL
LIN {X 0,Y 594.353,Z 260.759,A -85,B 0,C 180,E1 -1069.094,E2 -1069.094} C_VEL
LIN {X 0,Y 594.383,Z 260.757,A -85,B 0,C 180,E1 -1071.842,E2 -1071.842} C_VEL
LIN {X 0,Y 594.371,Z 260.753,A -85,B 0,C 180,E1 -1074.572,E2 -1074.572} C_VEL
LIN {X 0,Y 594.406,Z 260.757,A -85,B 0,C 180,E1 -1077.289,E2 -1077.289} C_VEL
LIN {X 0,Y 594.414,Z 260.749,A -85,B 0,C 180,E1 -1080,E2 -1080} C_VEL
LIN {X 0,Y 594.389,Z 260.753,A -85,B 0,C 180,E1 -1082.71,E2 -1082.71} C_VEL
LIN {X 0,Y 594.399,Z 260.759,A -85,B 0,C 180,E1 -1085.427,E2 -1085.427} C_VEL
LIN {X 0,Y 594.412,Z 260.748,A -85,B 0,C 180,E1 -1088.156,E2 -1088.156} C_VEL
LIN {X 0,Y 594.381,Z 260.76,A -85,B 0,C 180,E1 -1091.069,E2 -1091.069} C_VEL
LIN {X 0,Y 594.386,Z 260.756,A -85,B 0,C 180,E1 -1093.678,E2 -1093.678} C_VEL
LIN {X 0,Y 594.369,Z 260.757,A -85,B 0,C 180,E1 -1096.711,E2 -1096.711} C_VEL
LIN {X 0,Y 594.367,Z 260.763,A -85,B 0,C 180,E1 -1099.334,E2 -1099.334} C_VEL
LIN {X 0,Y 594.362,Z 260.76,A -85,B 0,C 180,E1 -1101.503,E2 -1101.503} C_VEL
LIN {X 0,Y 594.389,Z 260.753,A -85,B 0,C 180,E1 -1104.446,E2 -1104.446} C_VEL
LIN {X 0,Y 594.385,Z 260.757,A -85,B 0,C 180,E1 -1106.699,E2 -1106.699} C_VEL
LIN {X 0,Y 594.379,Z 260.762,A -85,B 0,C 180,E1 -1108.998,E2 -1108.998} C_VEL
LIN {X 0,Y 594.376,Z 260.755,A -85,B 0,C 180,E1 -1111.642,E2 -1111.642} C_VEL
LIN {X 0,Y 594.381,Z 260.757,A -85,B 0,C 180,E1 -1114.58,E2 -1114.58} C_VEL
LIN {X 0,Y 594.384,Z 260.761,A -85,B 0,C 180,E1 -1117.086,E2 -1117.086} C_VEL
LIN {X 0,Y 594.374,Z 260.754,A -85,B 0,C 180,E1 -1119.774,E2 -1119.774} C_VEL
LIN {X 0,Y 594.368,Z 260.757,A -85,B 0,C 180,E1 -1122.375,E2 -1122.375} C_VEL
LIN {X 0,Y 594.363,Z 260.761,A -85,B 0,C 180,E1 -1125.191,E2 -1125.191} C_VEL
LIN {X 0,Y 594.366,Z 260.755,A -85,B 0,C 180,E1 -1127.624,E2 -1127.624} C_VEL
LIN {X 0,Y 594.391,Z 260.755,A -85,B 0,C 180,E1 -1130.321,E2 -1130.321} C_VEL
LIN {X 0,Y 594.382,Z 260.761,A -85,B 0,C 180,E1 -1132.913,E2 -1132.913} C_VEL
LIN {X 0,Y 594.378,Z 260.754,A -85,B 0,C 180,E1 -1135.862,E2 -1135.862} C_VEL
LIN {X 0,Y 594.377,Z 260.764,A -85,B 0,C 180,E1 -1138.65,E2 -1138.65} C_VEL
LIN {X 0,Y 594.375,Z 260.761,A -85,B 0,C 180,E1 -1141.043,E2 -1141.043} C_VEL
LIN {X 0,Y 594.42,Z 260.945,A -85,B 0,C 180,E1 -1142.827,E2 -1142.827} C_VEL
LIN {X 0,Y 595.552,Z 265.361,A -85,B 0,C 180,E1 -1143.262,E2 -1143.262} C_VEL
LIN {X 0,Y 595.265,Z 298.486,A -85,B 0,C 180,E1 -1146.056,E2 -1146.056} C_VEL
LIN {X 0,Y 595.274,Z 312.395,A -85,B 0,C 180,E1 -1147.192,E2 -1147.192} C_VEL
LIN {X 0,Y 595.796,Z 317.075,A -85,B 0,C 180,E1 -1147.273,E2 -1147.273} C_VEL
LIN {X 0,Y 595.471,Z 517.94,A -85,B 0,C 180,E1 -1149.827,E2 -1149.827} C_VEL
LIN {X 0,Y 595.406,Z 534.176,A -85,B 0,C 180,E1 -1150.162,E2 -1150.162} C_VEL
LIN {X 0,Y 595.27,Z 550.943,A -85,B 0,C 180,E1 -1150.651,E2 -1150.651} C_VEL
LIN {X 0,Y 595.153,Z 566.485,A -85,B 0,C 180,E1 -1151.245,E2 -1151.245} C_VEL
LIN {X 0,Y 595.055,Z 581.017,A -85,B 0,C 180,E1 -1151.939,E2 -1151.939} C_VEL
LIN {X 0,Y 594.909,Z 594.846,A -85,B 0,C 180,E1 -1152.734,E2 -1152.734} C_VEL
LIN {X 0,Y 594.812,Z 609.052,A -85,B 0,C 180,E1 -1153.703,E2 -1153.703} C_VEL
LIN {X 0,Y 594.647,Z 622.125,A -85,B 0,C 180,E1 -1154.754,E2 -1154.754} C_VEL
LIN {X 0,Y 594.558,Z 634.315,A -85,B 0,C 180,E1 -1155.904,E2 -1155.904} C_VEL
LIN {X 0,Y 594.449,Z 645.911,A -85,B 0,C 180,E1 -1157.193,E2 -1157.193} C_VEL
LIN {X 0,Y 594.381,Z 656.423,A -85,B 0,C 180,E1 -1158.574,E2 -1158.574} C_VEL
LIN {X 0,Y 594.333,Z 665.273,A -85,B 0,C 180,E1 -1159.955,E2 -1159.955} C_VEL
LIN {X 0,Y 594.295,Z 673.487,A -85,B 0,C 180,E1 -1161.499,E2 -1161.499} C_VEL
LIN {X 0,Y 594.284,Z 679.468,A -85,B 0,C 180,E1 -1162.867,E2 -1162.867} C_VEL
LIN {X 0,Y 594.263,Z 685.246,A -85,B 0,C 180,E1 -1164.571,E2 -1164.571} C_VEL
LIN {X 0,Y 594.253,Z 688.634,A -85,B 0,C 180,E1 -1165.931,E2 -1165.931} C_VEL
LIN {X 0,Y 594.213,Z 691.087,A -85,B 0,C 180,E1 -1167.288,E2 -1167.288} C_VEL
LIN {X 0,Y 594.24,Z 692.478,A -85,B 0,C 180,E1 -1168.645,E2 -1168.645} C_VEL
LIN {X 0,Y 594.231,Z 693,A -85,B 0,C 180,E1 -1170,E2 -1170} C_VEL
LIN {X 0,Y 594.24,Z 692.478,A -85,B 0,C 180,E1 -1171.355,E2 -1171.355} C_VEL
LIN {X 0,Y 594.213,Z 691.087,A -85,B 0,C 180,E1 -1172.712,E2 -1172.712} C_VEL
LIN {X 0,Y 594.253,Z 688.633,A -85,B 0,C 180,E1 -1174.069,E2 -1174.069} C_VEL
LIN {X 0,Y 594.279,Z 684.185,A -85,B 0,C 180,E1 -1175.769,E2 -1175.769} C_VEL
LIN {X 0,Y 594.284,Z 679.468,A -85,B 0,C 180,E1 -1177.133,E2 -1177.133} C_VEL
LIN {X 0,Y 594.318,Z 671.857,A -85,B 0,C 180,E1 -1178.843,E2 -1178.843} C_VEL
LIN {X 0,Y 594.354,Z 663.247,A -85,B 0,C 180,E1 -1180.389,E2 -1180.389} C_VEL
LIN {X 0,Y 594.406,Z 653.969,A -85,B 0,C 180,E1 -1181.769,E2 -1181.769} C_VEL
LIN {X 0,Y 594.469,Z 644.422,A -85,B 0,C 180,E1 -1182.981,E2 -1182.981} C_VEL
LIN {X 0,Y 594.539,Z 632.948,A -85,B 0,C 180,E1 -1184.232,E2 -1184.232} C_VEL
LIN {X 0,Y 594.678,Z 621.142,A -85,B 0,C 180,E1 -1185.333,E2 -1185.333} C_VEL
LIN {X 0,Y 594.809,Z 607.881,A -85,B 0,C 180,E1 -1186.385,E2 -1186.385} C_VEL
LIN {X 0,Y 594.924,Z 593.432,A -85,B 0,C 180,E1 -1187.355,E2 -1187.355} C_VEL
LIN {X 0,Y 595.042,Z 579.264,A -85,B 0,C 180,E1 -1188.151,E2 -1188.151} C_VEL
LIN {X 0,Y 595.2,Z 564.109,A -85,B 0,C 180,E1 -1188.855,E2 -1188.855} C_VEL
LIN {X 0,Y 595.28,Z 548.342,A -85,B 0,C 180,E1 -1189.438,E2 -1189.438} C_VEL
LIN {X 0,Y 595.386,Z 532.346,A -85,B 0,C 180,E1 -1189.883,E2 -1189.883} C_VEL
LIN {X 0,Y 595.461,Z 516.425,A -85,B 0,C 180,E1 -1190.196,E2 -1190.196} C_VEL
LIN {X 0,Y 595.784,Z 315.458,A -85,B 0,C 180,E1 -1192.748,E2 -1192.748} C_VEL
LIN {X 0,Y 595.216,Z 312.027,A -85,B 0,C 180,E1 -1192.816,E2 -1192.816} C_VEL
LIN {X 0,Y 595.477,Z 276.401,A -85,B 0,C 180,E1 -1195.799,E2 -1195.799} C_VEL
LIN {X 0,Y 595.551,Z 265.359,A -85,B 0,C 180,E1 -1196.738,E2 -1196.738} C_VEL
LIN {X 0,Y 594.395,Z 260.761,A -85,B 0,C 180,E1 -1197.198,E2 -1197.198} C_VEL
LIN {X 0,Y 594.372,Z 260.758,A -85,B 0,C 180,E1 -1199.777,E2 -1199.777} C_VEL
LIN {X 0,Y 594.36,Z 260.757,A -85,B 0,C 180,E1 -1202.148,E2 -1202.148} C_VEL
LIN {X 0,Y 594.374,Z 260.756,A -85,B 0,C 180,E1 -1204.581,E2 -1204.581} C_VEL
LIN {X 0,Y 594.39,Z 260.756,A -85,B 0,C 180,E1 -1207.609,E2 -1207.609} C_VEL
LIN {X 0,Y 594.368,Z 260.757,A -85,B 0,C 180,E1 -1210.567,E2 -1210.567} C_VEL
LIN {X 0,Y 594.379,Z 260.76,A -85,B 0,C 180,E1 -1213.299,E2 -1213.299} C_VEL
LIN {X 0,Y 594.368,Z 260.755,A -85,B 0,C 180,E1 -1216.161,E2 -1216.161} C_VEL
LIN {X 0,Y 594.381,Z 260.755,A -85,B 0,C 180,E1 -1218.537,E2 -1218.537} C_VEL
LIN {X 0,Y 594.389,Z 260.757,A -85,B 0,C 180,E1 -1221.295,E2 -1221.295} C_VEL
LIN {X 0,Y 594.353,Z 260.757,A -85,B 0,C 180,E1 -1223.756,E2 -1223.756} C_VEL
LIN {X 0,Y 594.376,Z 260.754,A -85,B 0,C 180,E1 -1226.239,E2 -1226.239} C_VEL
LIN {X 0,Y 594.378,Z 260.759,A -85,B 0,C 180,E1 -1228.651,E2 -1228.651} C_VEL
LIN {X 0,Y 594.381,Z 260.758,A -85,B 0,C 180,E1 -1231.043,E2 -1231.043} C_VEL
LIN {X 0,Y 594.384,Z 260.753,A -85,B 0,C 180,E1 -1233.978,E2 -1233.978} C_VEL
LIN {X 0,Y 594.39,Z 260.754,A -85,B 0,C 180,E1 -1236.296,E2 -1236.296} C_VEL
LIN {X 0,Y 594.393,Z 260.754,A -85,B 0,C 180,E1 -1239.224,E2 -1239.224} C_VEL
LIN {X 0,Y 594.356,Z 260.757,A -85,B 0,C 180,E1 -1242.095,E2 -1242.095} C_VEL
LIN {X 0,Y 594.365,Z 260.757,A -85,B 0,C 180,E1 -1244.219,E2 -1244.219} C_VEL
LIN {X 0,Y 594.383,Z 260.757,A -85,B 0,C 180,E1 -1246.321,E2 -1246.321} C_VEL
LIN {X 0,Y 594.359,Z 260.757,A -85,B 0,C 180,E1 -1249.095,E2 -1249.095} C_VEL
LIN {X 0,Y 594.383,Z 260.753,A -85,B 0,C 180,E1 -1251.843,E2 -1251.843} C_VEL
LIN {X 0,Y 594.387,Z 260.76,A -85,B 0,C 180,E1 -1254.573,E2 -1254.573} C_VEL
LIN {X 0,Y 594.384,Z 260.753,A -85,B 0,C 180,E1 -1257.289,E2 -1257.289} C_VEL
LIN {X 0,Y 594.415,Z 260.752,A -85,B 0,C 180,E1 -1260,E2 -1260} C_VEL
LIN {X 0,Y 594.395,Z 260.756,A -85,B 0,C 180,E1 -1262.711,E2 -1262.711} C_VEL
LIN {X 0,Y 594.365,Z 260.755,A -85,B 0,C 180,E1 -1265.428,E2 -1265.428} C_VEL
LIN {X 0,Y 594.38,Z 260.759,A -85,B 0,C 180,E1 -1268.158,E2 -1268.158} C_VEL
LIN {X 0,Y 594.367,Z 260.755,A -85,B 0,C 180,E1 -1271.061,E2 -1271.061} C_VEL
LIN {X 0,Y 594.365,Z 260.755,A -85,B 0,C 180,E1 -1273.68,E2 -1273.68} C_VEL
LIN {X 0,Y 594.328,Z 260.759,A -85,B 0,C 180,E1 -1275.315,E2 -1275.315} C_VEL
LIN {X 0,Y 593.659,Z 260.848,A -85,B 0,C 180,E1 -1275.88,E2 -1275.88} C_VEL
LIN {X 0,Y 590.795,Z 261.21,A -85,B 0,C 180,E1 -1276.798,E2 -1276.798} C_VEL
LIN {X 0,Y 588.384,Z 261.513,A -85,B 0,C 180,E1 -1277.536,E2 -1277.536} C_VEL
LIN {X 0,Y 587.361,Z 261.636,A -85,B 0,C 180,E1 -1278.106,E2 -1278.106} C_VEL
LIN {X 0,Y 587.284,Z 261.643,A -85,B 0,C 180,E1 -1278.299,E2 -1278.299} C_VEL
LIN {X 0,Y 587.318,Z 261.633,A -85,B 0,C 180,E1 -1281.039,E2 -1281.039} C_VEL
LIN {X 0,Y 587.298,Z 261.643,A -85,B 0,C 180,E1 -1284.009,E2 -1284.009} C_VEL
LIN {X 0,Y 587.279,Z 261.645,A -85,B 0,C 180,E1 -1286.282,E2 -1286.282} C_VEL
LIN {X 0,Y 587.297,Z 261.635,A -85,B 0,C 180,E1 -1289.124,E2 -1289.124} C_VEL
LIN {X 0,Y 587.296,Z 261.643,A -85,B 0,C 180,E1 -1291.828,E2 -1291.828} C_VEL
LIN {X 0,Y 587.311,Z 261.638,A -85,B 0,C 180,E1 -1294.342,E2 -1294.342} C_VEL
LIN {X 0,Y 587.267,Z 261.64,A -85,B 0,C 180,E1 -1296.753,E2 -1296.753} C_VEL
LIN {X 0,Y 587.304,Z 261.637,A -85,B 0,C 180,E1 -1299.363,E2 -1299.363} C_VEL
LIN {X 0,Y 587.298,Z 261.642,A -85,B 0,C 180,E1 -1302.103,E2 -1302.103} C_VEL
LIN {X 0,Y 587.281,Z 261.639,A -85,B 0,C 180,E1 -1305.085,E2 -1305.085} C_VEL
LIN {X 0,Y 587.31,Z 261.643,A -85,B 0,C 180,E1 -1307.924,E2 -1307.924} C_VEL
LIN {X 0,Y 587.306,Z 261.638,A -85,B 0,C 180,E1 -1311.062,E2 -1311.062} C_VEL
LIN {X 0,Y 587.363,Z 261.834,A -85,B 0,C 180,E1 -1311.884,E2 -1311.884} C_VEL
LIN {X 0,Y 588.314,Z 265.767,A -85,B 0,C 180,E1 -1312.31,E2 -1312.31} C_VEL
LIN {X 0,Y 588.299,Z 282.374,A -85,B 0,C 180,E1 -1313.908,E2 -1313.908} C_VEL
LIN {X 0,Y 588.384,Z 283.522,A -85,B 0,C 180,E1 -1313.969,E2 -1313.969} C_VEL
LIN {X 0,Y 589.229,Z 288.294,A -85,B 0,C 180,E1 -1314.066,E2 -1314.066} C_VEL
LIN {X 0,Y 588.808,Z 489.406,A -85,B 0,C 180,E1 -1316.656,E2 -1316.656} C_VEL
LIN {X 0,Y 588.672,Z 506.191,A -85,B 0,C 180,E1 -1317.021,E2 -1317.021} C_VEL
LIN {X 0,Y 588.53,Z 521.776,A -85,B 0,C 180,E1 -1317.495,E2 -1317.495} C_VEL
LIN {X 0,Y 588.354,Z 537.643,A -85,B 0,C 180,E1 -1318.118,E2 -1318.118} C_VEL
LIN {X 0,Y 588.207,Z 553.22,A -85,B 0,C 180,E1 -1318.885,E2 -1318.885} C_VEL
LIN {X 0,Y 588.012,Z 568.403,A -85,B 0,C 180,E1 -1319.796,E2 -1319.796} C_VEL
LIN {X 0,Y 587.843,Z 582.078,A -85,B 0,C 180,E1 -1320.782,E2 -1320.782} C_VEL
LIN {X 0,Y 587.68,Z 595.35,A -85,B 0,C 180,E1 -1321.908,E2 -1321.908} C_VEL
LIN {X 0,Y 587.551,Z 607.827,A -85,B 0,C 180,E1 -1323.157,E2 -1323.157} C_VEL
LIN {X 0,Y 587.413,Z 619.113,A -85,B 0,C 180,E1 -1324.487,E2 -1324.487} C_VEL
LIN {X 0,Y 587.348,Z 627.995,A -85,B 0,C 180,E1 -1325.706,E2 -1325.706} C_VEL
LIN {X 0,Y 587.264,Z 636.827,A -85,B 0,C 180,E1 -1327.146,E2 -1327.146} C_VEL
LIN {X 0,Y 587.234,Z 644.186,A -85,B 0,C 180,E1 -1328.591,E2 -1328.591} C_VEL
LIN {X 0,Y 587.189,Z 650.303,A -85,B 0,C 180,E1 -1330.055,E2 -1330.055} C_VEL
LIN {X 0,Y 587.161,Z 655.113,A -85,B 0,C 180,E1 -1331.507,E2 -1331.507} C_VEL
LIN {X 0,Y 587.13,Z 657.922,A -85,B 0,C 180,E1 -1332.587,E2 -1332.587} C_VEL
LIN {X 0,Y 587.134,Z 660.636,A -85,B 0,C 180,E1 -1334.019,E2 -1334.019} C_VEL
LIN {X 0,Y 587.162,Z 662.578,A -85,B 0,C 180,E1 -1335.82,E2 -1335.82} C_VEL
LIN {X 0,Y 587.14,Z 662.963,A -85,B 0,C 180,E1 -1336.854,E2 -1336.854} C_VEL
LIN {X 0,Y 587.152,Z 662.586,A -85,B 0,C 180,E1 -1338.259,E2 -1338.259} C_VEL
LIN {X 0,Y 587.137,Z 661.257,A -85,B 0,C 180,E1 -1339.656,E2 -1339.656} C_VEL
LIN {X 0,Y 587.125,Z 658.877,A -85,B 0,C 180,E1 -1341.048,E2 -1341.048} C_VEL
LIN {X 0,Y 587.146,Z 655.55,A -85,B 0,C 180,E1 -1342.434,E2 -1342.434} C_VEL
LIN {X 0,Y 587.181,Z 651.088,A -85,B 0,C 180,E1 -1343.816,E2 -1343.816} C_VEL
LIN {X 0,Y 587.225,Z 645.606,A -85,B 0,C 180,E1 -1345.194,E2 -1345.194} C_VEL
LIN {X 0,Y 587.21,Z 638.867,A -85,B 0,C 180,E1 -1346.569,E2 -1346.569} C_VEL
LIN {X 0,Y 587.317,Z 630.834,A -85,B 0,C 180,E1 -1347.943,E2 -1347.943} C_VEL
LIN {X 0,Y 587.401,Z 621.349,A -85,B 0,C 180,E1 -1349.314,E2 -1349.314} C_VEL
LIN {X 0,Y 587.496,Z 610.125,A -85,B 0,C 180,E1 -1350.685,E2 -1350.685} C_VEL
LIN {X 0,Y 587.632,Z 598.555,A -85,B 0,C 180,E1 -1351.885,E2 -1351.885} C_VEL
LIN {X 0,Y 587.805,Z 585.951,A -85,B 0,C 180,E1 -1352.998,E2 -1352.998} C_VEL
LIN {X 0,Y 587.93,Z 572.306,A -85,B 0,C 180,E1 -1354.027,E2 -1354.027} C_VEL
LIN {X 0,Y 588.129,Z 557.381,A -85,B 0,C 180,E1 -1354.97,E2 -1354.97} C_VEL
LIN {X 0,Y 588.315,Z 542.691,A -85,B 0,C 180,E1 -1355.742,E2 -1355.742} C_VEL
LIN {X 0,Y 588.515,Z 526.515,A -85,B 0,C 180,E1 -1356.428,E2 -1356.428} C_VEL
LIN {X 0,Y 588.674,Z 509.783,A -85,B 0,C 180,E1 -1356.971,E2 -1356.971} C_VEL
LIN {X 0,Y 588.782,Z 493.493,A -85,B 0,C 180,E1 -1357.354,E2 -1357.354} C_VEL
LIN {X 0,Y 588.848,Z 472.188,A -85,B 0,C 180,E1 -1357.673,E2 -1357.673} C_VEL
LIN {X 0,Y 589.209,Z 287.473,A -85,B 0,C 180,E1 -1360.035,E2 -1360.035} C_VEL
LIN {X 0,Y 588.319,Z 282.718,A -85,B 0,C 180,E1 -1360.149,E2 -1360.149} C_VEL
LIN {X 0,Y 588.415,Z 266.394,A -85,B 0,C 180,E1 -1361.715,E2 -1361.715} C_VEL
LIN {X 0,Y 587.34,Z 261.639,A -85,B 0,C 180,E1 -1362.241,E2 -1362.241} C_VEL
LIN {X 0,Y 587.333,Z 261.639,A -85,B 0,C 180,E1 -1364.554,E2 -1364.554} C_VEL
LIN {X 0,Y 587.278,Z 261.638,A -85,B 0,C 180,E1 -1367.408,E2 -1367.408} C_VEL
LIN {X 0,Y 587.302,Z 261.637,A -85,B 0,C 180,E1 -1369.576,E2 -1369.576} C_VEL
LIN {X 0,Y 587.305,Z 261.638,A -85,B 0,C 180,E1 -1371.775,E2 -1371.775} C_VEL
LIN {X 0,Y 587.309,Z 261.636,A -85,B 0,C 180,E1 -1374.76,E2 -1374.76} C_VEL
LIN {X 0,Y 587.288,Z 261.64,A -85,B 0,C 180,E1 -1377.68,E2 -1377.68} C_VEL
LIN {X 0,Y 587.315,Z 261.638,A -85,B 0,C 180,E1 -1380.505,E2 -1380.505} C_VEL
LIN {X 0,Y 587.306,Z 261.636,A -85,B 0,C 180,E1 -1383.399,E2 -1383.399} C_VEL
LIN {X 0,Y 587.27,Z 261.646,A -85,B 0,C 180,E1 -1385.902,E2 -1385.902} C_VEL
LIN {X 0,Y 587.273,Z 261.641,A -85,B 0,C 180,E1 -1388.484,E2 -1388.484} C_VEL
LIN {X 0,Y 587.282,Z 261.637,A -85,B 0,C 180,E1 -1391.162,E2 -1391.162} C_VEL
LIN {X 0,Y 587.286,Z 261.645,A -85,B 0,C 180,E1 -1394.109,E2 -1394.109} C_VEL
LIN {X 0,Y 587.274,Z 261.637,A -85,B 0,C 180,E1 -1396.989,E2 -1396.989} C_VEL
LIN {X 0,Y 587.293,Z 261.644,A -85,B 0,C 180,E1 -1399.985,E2 -1399.985} C_VEL
LIN {X 0,Y 587.309,Z 261.632,A -85,B 0,C 180,E1 -1402.389,E2 -1402.389} C_VEL
LIN {X 0,Y 587.327,Z 261.637,A -85,B 0,C 180,E1 -1405.655,E2 -1405.655} C_VEL
LIN {X 0,Y 587.334,Z 261.634,A -85,B 0,C 180,E1 -1408.23,E2 -1408.23} C_VEL
LIN {X 0,Y 587.3,Z 261.634,A -85,B 0,C 180,E1 -1410.875,E2 -1410.875} C_VEL
LIN {X 0,Y 587.303,Z 261.643,A -85,B 0,C 180,E1 -1413.83,E2 -1413.83} C_VEL
LIN {X 0,Y 587.317,Z 261.637,A -85,B 0,C 180,E1 -1415.992,E2 -1415.992} C_VEL
LIN {X 0,Y 587.311,Z 261.636,A -85,B 0,C 180,E1 -1418.225,E2 -1418.225} C_VEL
LIN {X 0,Y 587.334,Z 261.633,A -85,B 0,C 180,E1 -1421.15,E2 -1421.15} C_VEL
LIN {X 0,Y 587.304,Z 261.638,A -85,B 0,C 180,E1 -1424.024,E2 -1424.024} C_VEL
LIN {X 0,Y 587.351,Z 261.63,A -85,B 0,C 180,E1 -1426.154,E2 -1426.154} C_VEL
LIN {X 0,Y 587.339,Z 261.631,A -85,B 0,C 180,E1 -1428.962,E2 -1428.962} C_VEL
LIN {X 0,Y 587.342,Z 261.636,A -85,B 0,C 180,E1 -1431.744,E2 -1431.744} C_VEL
LIN {X 0,Y 587.323,Z 261.636,A -85,B 0,C 180,E1 -1433.817,E2 -1433.817} C_VEL
LIN {X 0,Y 587.315,Z 261.637,A -85,B 0,C 180,E1 -1435.882,E2 -1435.882} C_VEL
LIN {X 0,Y 587.374,Z 261.628,A -85,B 0,C 180,E1 -1437.943,E2 -1437.943} C_VEL
LIN {X 0,Y 587.374,Z 261.625,A -85,B 0,C 180,E1 -1440.685,E2 -1440.685} C_VEL
LIN {X 0,Y 587.331,Z 261.641,A -85,B 0,C 180,E1 -1443.43,E2 -1443.43} C_VEL
LIN {X 0,Y 587.329,Z 261.63,A -85,B 0,C 180,E1 -1446.182,E2 -1446.182} C_VEL
LIN {X 0,Y 587.363,Z 261.626,A -85,B 0,C 180,E1 -1448.255,E2 -1448.255} C_VEL
LIN {X 0,Y 587.349,Z 261.637,A -85,B 0,C 180,E1 -1451.133,E2 -1451.133} C_VEL
LIN {X 0,Y 587.362,Z 261.629,A -85,B 0,C 180,E1 -1453.845,E2 -1453.845} C_VEL
LIN {X 0,Y 587.339,Z 261.634,A -85,B 0,C 180,E1 -1456.81,E2 -1456.81} C_VEL
LIN {X 0,Y 587.314,Z 261.637,A -85,B 0,C 180,E1 -1459.576,E2 -1459.576} C_VEL
LIN {X 0,Y 587.338,Z 261.631,A -85,B 0,C 180,E1 -1462.514,E2 -1462.514} C_VEL
LIN {X 0,Y 587.351,Z 261.633,A -85,B 0,C 180,E1 -1464.758,E2 -1464.758} C_VEL
LIN {X 0,Y 587.351,Z 261.63,A -85,B 0,C 180,E1 -1467.693,E2 -1467.693} C_VEL
LIN {X 0,Y 587.336,Z 261.633,A -85,B 0,C 180,E1 -1470.51,E2 -1470.51} C_VEL
LIN {X 0,Y 587.332,Z 261.635,A -85,B 0,C 180,E1 -1473.396,E2 -1473.396} C_VEL
LIN {X 0,Y 587.312,Z 261.633,A -85,B 0,C 180,E1 -1475.898,E2 -1475.898} C_VEL
LIN {X 0,Y 587.334,Z 261.634,A -85,B 0,C 180,E1 -1478.479,E2 -1478.479} C_VEL
LIN {X 0,Y 587.335,Z 261.637,A -85,B 0,C 180,E1 -1481.157,E2 -1481.157} C_VEL
LIN {X 0,Y 587.325,Z 261.632,A -85,B 0,C 180,E1 -1484.113,E2 -1484.113} C_VEL
LIN {X 0,Y 587.319,Z 261.641,A -85,B 0,C 180,E1 -1486.994,E2 -1486.994} C_VEL
LIN {X 0,Y 587.316,Z 261.633,A -85,B 0,C 180,E1 -1489.746,E2 -1489.746} C_VEL
LIN {X 0,Y 587.344,Z 261.634,A -85,B 0,C 180,E1 -1492.392,E2 -1492.392} C_VEL
LIN {X 0,Y 587.344,Z 261.63,A -85,B 0,C 180,E1 -1495.653,E2 -1495.653} C_VEL
LIN {X 0,Y 587.342,Z 261.634,A -85,B 0,C 180,E1 -1498.231,E2 -1498.231} C_VEL
LIN {X 0,Y 587.343,Z 261.64,A -85,B 0,C 180,E1 -1500.867,E2 -1500.867} C_VEL
LIN {X 0,Y 587.362,Z 261.801,A -85,B 0,C 180,E1 -1502.548,E2 -1502.548} C_VEL
LIN {X 0,Y 588.686,Z 266.465,A -85,B 0,C 180,E1 -1503.021,E2 -1503.021} C_VEL
LIN {X 0,Y 588.858,Z 273.993,A -85,B 0,C 180,E1 -1503.682,E2 -1503.682} C_VEL
LIN {X 0,Y 588.507,Z 309.528,A -85,B 0,C 180,E1 -1506.698,E2 -1506.698} C_VEL
LIN {X 0,Y 588.489,Z 311.978,A -85,B 0,C 180,E1 -1506.904,E2 -1506.904} C_VEL
LIN {X 0,Y 589.248,Z 317.673,A -85,B 0,C 180,E1 -1507.014,E2 -1507.014} C_VEL
LIN {X 0,Y 588.806,Z 517.94,A -85,B 0,C 180,E1 -1509.589,E2 -1509.589} C_VEL
LIN {X 0,Y 588.706,Z 534.177,A -85,B 0,C 180,E1 -1509.927,E2 -1509.927} C_VEL
LIN {X 0,Y 588.547,Z 550.945,A -85,B 0,C 180,E1 -1510.421,E2 -1510.421} C_VEL
LIN {X 0,Y 588.406,Z 566.722,A -85,B 0,C 180,E1 -1511.033,E2 -1511.033} C_VEL
LIN {X 0,Y 588.248,Z 581.02,A -85,B 0,C 180,E1 -1511.723,E2 -1511.723} C_VEL
LIN {X 0,Y 588.076,Z 594.849,A -85,B 0,C 180,E1 -1512.527,E2 -1512.527} C_VEL
LIN {X 0,Y 587.916,Z 609.054,A -85,B 0,C 180,E1 -1513.506,E2 -1513.506} C_VEL
LIN {X 0,Y 587.729,Z 622.124,A -85,B 0,C 180,E1 -1514.57,E2 -1514.57} C_VEL
LIN {X 0,Y 587.563,Z 633.627,A -85,B 0,C 180,E1 -1515.663,E2 -1515.663} C_VEL
LIN {X 0,Y 587.449,Z 644.424,A -85,B 0,C 180,E1 -1516.861,E2 -1516.861} C_VEL
LIN {X 0,Y 587.351,Z 655.21,A -85,B 0,C 180,E1 -1518.263,E2 -1518.263} C_VEL
LIN {X 0,Y 587.297,Z 664.261,A -85,B 0,C 180,E1 -1519.659,E2 -1519.659} C_VEL
LIN {X 0,Y 587.245,Z 671.857,A -85,B 0,C 180,E1 -1521.05,E2 -1521.05} C_VEL
LIN {X 0,Y 587.207,Z 679.468,A -85,B 0,C 180,E1 -1522.781,E2 -1522.781} C_VEL
LIN {X 0,Y 587.187,Z 685.247,A -85,B 0,C 180,E1 -1524.506,E2 -1524.506} C_VEL
LIN {X 0,Y 587.168,Z 688.635,A -85,B 0,C 180,E1 -1525.882,E2 -1525.882} C_VEL
LIN {X 0,Y 587.119,Z 691.088,A -85,B 0,C 180,E1 -1527.256,E2 -1527.256} C_VEL
LIN {X 0,Y 587.14,Z 692.478,A -85,B 0,C 180,E1 -1528.628,E2 -1528.628} C_VEL
LIN {X 0,Y 587.132,Z 693,A -85,B 0,C 180,E1 -1530,E2 -1530} C_VEL
LIN {X 0,Y 587.14,Z 692.478,A -85,B 0,C 180,E1 -1531.372,E2 -1531.372} C_VEL
LIN {X 0,Y 587.119,Z 691.087,A -85,B 0,C 180,E1 -1532.745,E2 -1532.745} C_VEL
LIN {X 0,Y 587.168,Z 688.634,A -85,B 0,C 180,E1 -1534.118,E2 -1534.118} C_VEL
LIN {X 0,Y 587.187,Z 684.186,A -85,B 0,C 180,E1 -1535.839,E2 -1535.839} C_VEL
LIN {X 0,Y 587.207,Z 679.468,A -85,B 0,C 180,E1 -1537.22,E2 -1537.22} C_VEL
LIN {X 0,Y 587.245,Z 671.857,A -85,B 0,C 180,E1 -1538.951,E2 -1538.951} C_VEL
LIN {X 0,Y 587.302,Z 663.248,A -85,B 0,C 180,E1 -1540.515,E2 -1540.515} C_VEL
LIN {X 0,Y 587.366,Z 653.97,A -85,B 0,C 180,E1 -1541.912,E2 -1541.912} C_VEL
LIN {X 0,Y 587.449,Z 644.423,A -85,B 0,C 180,E1 -1543.139,E2 -1543.139} C_VEL
LIN {X 0,Y 587.589,Z 632.568,A -85,B 0,C 180,E1 -1544.441,E2 -1544.441} C_VEL
LIN {X 0,Y 587.759,Z 620.094,A -85,B 0,C 180,E1 -1545.607,E2 -1545.607} C_VEL
LIN {X 0,Y 587.909,Z 606.704,A -85,B 0,C 180,E1 -1546.673,E2 -1546.673} C_VEL
LIN {X 0,Y 588.087,Z 592.005,A -85,B 0,C 180,E1 -1547.653,E2 -1547.653} C_VEL
LIN {X 0,Y 588.257,Z 577.519,A -85,B 0,C 180,E1 -1548.458,E2 -1548.458} C_VEL
LIN {X 0,Y 588.445,Z 562.39,A -85,B 0,C 180,E1 -1549.149,E2 -1549.149} C_VEL
LIN {X 0,Y 588.617,Z 546.244,A -85,B 0,C 180,E1 -1549.735,E2 -1549.735} C_VEL
LIN {X 0,Y 588.754,Z 529.598,A -85,B 0,C 180,E1 -1550.185,E2 -1550.185} C_VEL
LIN {X 0,Y 588.797,Z 513.412,A -85,B 0,C 180,E1 -1550.48,E2 -1550.48} C_VEL
LIN {X 0,Y 589.25,Z 316.682,A -85,B 0,C 180,E1 -1552.999,E2 -1552.999} C_VEL
LIN {X 0,Y 588.479,Z 312.006,A -85,B 0,C 180,E1 -1553.094,E2 -1553.094} C_VEL
LIN {X 0,Y 588.827,Z 276.401,A -85,B 0,C 180,E1 -1556.112,E2 -1556.112} C_VEL
LIN {X 0,Y 588.899,Z 268.345,A -85,B 0,C 180,E1 -1556.805,E2 -1556.805} C_VEL
LIN {X 0,Y 588.07,Z 264.271,A -85,B 0,C 180,E1 -1557.2,E2 -1557.2} C_VEL
LIN {X 0,Y 587.352,Z 261.639,A -85,B 0,C 180,E1 -1557.475,E2 -1557.475} C_VEL
LIN {X 0,Y 587.332,Z 261.633,A -85,B 0,C 180,E1 -1560.17,E2 -1560.17} C_VEL
LIN {X 0,Y 587.334,Z 261.633,A -85,B 0,C 180,E1 -1562.579,E2 -1562.579} C_VEL
LIN {X 0,Y 587.321,Z 261.641,A -85,B 0,C 180,E1 -1565.056,E2 -1565.056} C_VEL
LIN {X 0,Y 587.34,Z 261.632,A -85,B 0,C 180,E1 -1567.839,E2 -1567.839} C_VEL
LIN {X 0,Y 587.317,Z 261.633,A -85,B 0,C 180,E1 -1570.254,E2 -1570.254} C_VEL
LIN {X 0,Y 587.32,Z 261.64,A -85,B 0,C 180,E1 -1573.006,E2 -1573.006} C_VEL
LIN {X 0,Y 587.326,Z 261.632,A -85,B 0,C 180,E1 -1575.887,E2 -1575.887} C_VEL
LIN {X 0,Y 587.337,Z 261.637,A -85,B 0,C 180,E1 -1578.844,E2 -1578.844} C_VEL
LIN {X 0,Y 587.334,Z 261.633,A -85,B 0,C 180,E1 -1581.521,E2 -1581.521} C_VEL
LIN {X 0,Y 587.292,Z 261.636,A -85,B 0,C 180,E1 -1584.1,E2 -1584.1} C_VEL
LIN {X 0,Y 587.333,Z 261.635,A -85,B 0,C 180,E1 -1586.604,E2 -1586.604} C_VEL
LIN {X 0,Y 587.337,Z 261.632,A -85,B 0,C 180,E1 -1589.491,E2 -1589.491} C_VEL
LIN {X 0,Y 587.352,Z 261.629,A -85,B 0,C 180,E1 -1592.308,E2 -1592.308} C_VEL
LIN {X 0,Y 587.352,Z 261.632,A -85,B 0,C 180,E1 -1595.242,E2 -1595.242} C_VEL
LIN {X 0,Y 587.318,Z 261.633,A -85,B 0,C 180,E1 -1598.226,E2 -1598.226} C_VEL
LIN {X 0,Y 587.343,Z 261.633,A -85,B 0,C 180,E1 -1601.151,E2 -1601.151} C_VEL
LIN {X 0,Y 587.325,Z 261.631,A -85,B 0,C 180,E1 -1603.311,E2 -1603.311} C_VEL
LIN {X 0,Y 587.361,Z 261.63,A -85,B 0,C 180,E1 -1606.155,E2 -1606.155} C_VEL
LIN {X 0,Y 587.339,Z 261.632,A -85,B 0,C 180,E1 -1608.963,E2 -1608.963} C_VEL
LIN {X 0,Y 587.342,Z 261.63,A -85,B 0,C 180,E1 -1611.745,E2 -1611.745} C_VEL
LIN {X 0,Y 587.353,Z 261.637,A -85,B 0,C 180,E1 -1614.507,E2 -1614.507} C_VEL
LIN {X 0,Y 587.353,Z 261.629,A -85,B 0,C 180,E1 -1617.257,E2 -1617.257} C_VEL
LIN {X 0,Y 587.384,Z 261.628,A -85,B 0,C 180,E1 -1620,E2 -1620} C_VEL
LIN {X 0,Y 587.36,Z 261.632,A -85,B 0,C 180,E1 -1622.744,E2 -1622.744} C_VEL
LIN {X 0,Y 587.333,Z 261.631,A -85,B 0,C 180,E1 -1625.494,E2 -1625.494} C_VEL
LIN {X 0,Y 587.339,Z 261.637,A -85,B 0,C 180,E1 -1628.256,E2 -1628.256} C_VEL
LIN {X 0,Y 587.334,Z 261.631,A -85,B 0,C 180,E1 -1631.125,E2 -1631.125} C_VEL
LIN {X 0,Y 587.349,Z 261.631,A -85,B 0,C 180,E1 -1633.846,E2 -1633.846} C_VEL
LIN {X 0,Y 587.294,Z 261.638,A -85,B 0,C 180,E1 -1636.795,E2 -1636.795} C_VEL
LIN {X 0,Y 587.284,Z 261.643,A -85,B 0,C 180,E1 -1638.299,E2 -1638.299} C_VEL
LIN {X 0,Y 586.646,Z 261.717,A -85,B 0,C 180,E1 -1638.871,E2 -1638.871} C_VEL
LIN {X 0,Y 583.838,Z 262.068,A -85,B 0,C 180,E1 -1639.8,E2 -1639.8} C_VEL
LIN {X 0,Y 581.435,Z 262.37,A -85,B 0,C 180,E1 -1640.547,E2 -1640.547} C_VEL
LIN {X 0,Y 580.375,Z 262.498,A -85,B 0,C 180,E1 -1641.123,E2 -1641.123} C_VEL
LIN {X 0,Y 580.275,Z 262.511,A -85,B 0,C 180,E1 -1641.318,E2 -1641.318} C_VEL
LIN {X 0,Y 580.262,Z 262.519,A -85,B 0,C 180,E1 -1644.318,E2 -1644.318} C_VEL
LIN {X 0,Y 580.225,Z 262.519,A -85,B 0,C 180,E1 -1646.626,E2 -1646.626} C_VEL
LIN {X 0,Y 580.25,Z 262.513,A -85,B 0,C 180,E1 -1649.3,E2 -1649.3} C_VEL
LIN {X 0,Y 580.27,Z 262.518,A -85,B 0,C 180,E1 -1652.203,E2 -1652.203} C_VEL
LIN {X 0,Y 580.261,Z 262.513,A -85,B 0,C 180,E1 -1654.699,E2 -1654.699} C_VEL
LIN {X 0,Y 580.269,Z 262.519,A -85,B 0,C 180,E1 -1658.07,E2 -1658.07} C_VEL
LIN {X 0,Y 580.237,Z 262.515,A -85,B 0,C 180,E1 -1660.849,E2 -1660.849} C_VEL
LIN {X 0,Y 580.228,Z 262.524,A -85,B 0,C 180,E1 -1663.663,E2 -1663.663} C_VEL
LIN {X 0,Y 580.237,Z 262.518,A -85,B 0,C 180,E1 -1666.338,E2 -1666.338} C_VEL
LIN {X 0,Y 580.241,Z 262.517,A -85,B 0,C 180,E1 -1669.151,E2 -1669.151} C_VEL
LIN {X 0,Y 580.305,Z 262.632,A -85,B 0,C 180,E1 -1671.636,E2 -1671.636} C_VEL
LIN {X 0,Y 581.649,Z 268.41,A -85,B 0,C 180,E1 -1672.266,E2 -1672.266} C_VEL
LIN {X 0,Y 581.535,Z 282.773,A -85,B 0,C 180,E1 -1673.661,E2 -1673.661} C_VEL
LIN {X 0,Y 582.698,Z 289.273,A -85,B 0,C 180,E1 -1673.806,E2 -1673.806} C_VEL
LIN {X 0,Y 582.164,Z 489.035,A -85,B 0,C 180,E1 -1676.407,E2 -1676.407} C_VEL
LIN {X 0,Y 581.989,Z 504.962,A -85,B 0,C 180,E1 -1676.75,E2 -1676.75} C_VEL
LIN {X 0,Y 581.863,Z 520.841,A -85,B 0,C 180,E1 -1677.228,E2 -1677.228} C_VEL
LIN {X 0,Y 581.676,Z 536.008,A -85,B 0,C 180,E1 -1677.817,E2 -1677.817} C_VEL
LIN {X 0,Y 581.454,Z 549.794,A -85,B 0,C 180,E1 -1678.482,E2 -1678.482} C_VEL
LIN {X 0,Y 581.268,Z 563.532,A -85,B 0,C 180,E1 -1679.276,E2 -1679.276} C_VEL
LIN {X 0,Y 581.017,Z 576.699,A -85,B 0,C 180,E1 -1680.168,E2 -1680.168} C_VEL
LIN {X 0,Y 580.804,Z 591.276,A -85,B 0,C 180,E1 -1681.348,E2 -1681.348} C_VEL
LIN {X 0,Y 580.605,Z 604.426,A -85,B 0,C 180,E1 -1682.614,E2 -1682.614} C_VEL
LIN {X 0,Y 580.429,Z 616.563,A -85,B 0,C 180,E1 -1684.002,E2 -1684.002} C_VEL
LIN {X 0,Y 580.335,Z 625.935,A -85,B 0,C 180,E1 -1685.268,E2 -1685.268} C_VEL
LIN {X 0,Y 580.219,Z 635.329,A -85,B 0,C 180,E1 -1686.763,E2 -1686.763} C_VEL
LIN {X 0,Y 580.138,Z 643.399,A -85,B 0,C 180,E1 -1688.316,E2 -1688.316} C_VEL
LIN {X 0,Y 580.104,Z 649.706,A -85,B 0,C 180,E1 -1689.801,E2 -1689.801} C_VEL
LIN {X 0,Y 580.066,Z 654.622,A -85,B 0,C 180,E1 -1691.277,E2 -1691.277} C_VEL
LIN {X 0,Y 580.044,Z 657.537,A -85,B 0,C 180,E1 -1692.368,E2 -1692.368} C_VEL
LIN {X 0,Y 580.031,Z 660.376,A -85,B 0,C 180,E1 -1693.818,E2 -1693.818} C_VEL
LIN {X 0,Y 580.008,Z 662.206,A -85,B 0,C 180,E1 -1695.258,E2 -1695.258} C_VEL
LIN {X 0,Y 580.056,Z 662.927,A -85,B 0,C 180,E1 -1696.691,E2 -1696.691} C_VEL
LIN {X 0,Y 580.051,Z 662.694,A -85,B 0,C 180,E1 -1698.113,E2 -1698.113} C_VEL
LIN {X 0,Y 580.057,Z 661.44,A -85,B 0,C 180,E1 -1699.529,E2 -1699.529} C_VEL
LIN {X 0,Y 580.025,Z 659.207,A -85,B 0,C 180,E1 -1700.937,E2 -1700.937} C_VEL
LIN {X 0,Y 580.067,Z 655.958,A -85,B 0,C 180,E1 -1702.341,E2 -1702.341} C_VEL
LIN {X 0,Y 580.094,Z 651.652,A -85,B 0,C 180,E1 -1703.74,E2 -1703.74} C_VEL
LIN {X 0,Y 580.126,Z 646.291,A -85,B 0,C 180,E1 -1705.135,E2 -1705.135} C_VEL
LIN {X 0,Y 580.137,Z 639.69,A -85,B 0,C 180,E1 -1706.527,E2 -1706.527} C_VEL
LIN {X 0,Y 580.27,Z 630.742,A -85,B 0,C 180,E1 -1708.091,E2 -1708.091} C_VEL
LIN {X 0,Y 580.366,Z 621.241,A -85,B 0,C 180,E1 -1709.48,E2 -1709.48} C_VEL
LIN {X 0,Y 580.494,Z 609.998,A -85,B 0,C 180,E1 -1710.867,E2 -1710.867} C_VEL
LIN {X 0,Y 580.7,Z 598.409,A -85,B 0,C 180,E1 -1712.081,E2 -1712.081} C_VEL
LIN {X 0,Y 580.902,Z 585.778,A -85,B 0,C 180,E1 -1713.208,E2 -1713.208} C_VEL
LIN {X 0,Y 581.083,Z 572.097,A -85,B 0,C 180,E1 -1714.248,E2 -1714.248} C_VEL
LIN {X 0,Y 581.307,Z 557.132,A -85,B 0,C 180,E1 -1715.202,E2 -1715.202} C_VEL
LIN {X 0,Y 581.549,Z 542.365,A -85,B 0,C 180,E1 -1715.983,E2 -1715.983} C_VEL
LIN {X 0,Y 581.782,Z 527.208,A -85,B 0,C 180,E1 -1716.633,E2 -1716.633} C_VEL
LIN {X 0,Y 581.973,Z 510.933,A -85,B 0,C 180,E1 -1717.176,E2 -1717.176} C_VEL
LIN {X 0,Y 582.124,Z 494.478,A -85,B 0,C 180,E1 -1717.577,E2 -1717.577} C_VEL
LIN {X 0,Y 582.207,Z 476.817,A -85,B 0,C 180,E1 -1717.859,E2 -1717.859} C_VEL
LIN {X 0,Y 582.682,Z 288.717,A -85,B 0,C 180,E1 -1720.292,E2 -1720.292} C_VEL
LIN {X 0,Y 581.567,Z 282.831,A -85,B 0,C 180,E1 -1720.422,E2 -1720.422} C_VEL
LIN {X 0,Y 581.645,Z 268.11,A -85,B 0,C 180,E1 -1721.853,E2 -1721.853} C_VEL
LIN {X 0,Y 580.28,Z 262.519,A -85,B 0,C 180,E1 -1722.481,E2 -1722.481} C_VEL
LIN {X 0,Y 580.279,Z 262.515,A -85,B 0,C 180,E1 -1724.734,E2 -1724.734} C_VEL
LIN {X 0,Y 580.245,Z 262.516,A -85,B 0,C 180,E1 -1727.626,E2 -1727.626} C_VEL
LIN {X 0,Y 580.278,Z 262.514,A -85,B 0,C 180,E1 -1729.823,E2 -1729.823} C_VEL
LIN {X 0,Y 580.279,Z 262.513,A -85,B 0,C 180,E1 -1732.803,E2 -1732.803} C_VEL
LIN {X 0,Y 580.248,Z 262.514,A -85,B 0,C 180,E1 -1735.082,E2 -1735.082} C_VEL
LIN {X 0,Y 580.236,Z 262.521,A -85,B 0,C 180,E1 -1737.846,E2 -1737.846} C_VEL
LIN {X 0,Y 580.259,Z 262.515,A -85,B 0,C 180,E1 -1740.689,E2 -1740.689} C_VEL
LIN {X 0,Y 580.268,Z 262.512,A -85,B 0,C 180,E1 -1743.31,E2 -1743.31} C_VEL
LIN {X 0,Y 580.217,Z 262.522,A -85,B 0,C 180,E1 -1745.751,E2 -1745.751} C_VEL
LIN {X 0,Y 580.235,Z 262.523,A -85,B 0,C 180,E1 -1748.15,E2 -1748.15} C_VEL
LIN {X 0,Y 580.233,Z 262.515,A -85,B 0,C 180,E1 -1750.849,E2 -1750.849} C_VEL
LIN {X 0,Y 580.224,Z 262.521,A -85,B 0,C 180,E1 -1753.663,E2 -1753.663} C_VEL
LIN {X 0,Y 580.223,Z 262.517,A -85,B 0,C 180,E1 -1756.615,E2 -1756.615} C_VEL
LIN {X 0,Y 580.236,Z 262.516,A -85,B 0,C 180,E1 -1759.151,E2 -1759.151} C_VEL
LIN {X 0,Y 580.278,Z 262.514,A -85,B 0,C 180,E1 -1761.929,E2 -1761.929} C_VEL
LIN {X 0,Y 580.271,Z 262.51,A -85,B 0,C 180,E1 -1765.302,E2 -1765.302} C_VEL
LIN {X 0,Y 580.283,Z 262.516,A -85,B 0,C 180,E1 -1767.972,E2 -1767.972} C_VEL
LIN {X 0,Y 580.253,Z 262.511,A -85,B 0,C 180,E1 -1770.699,E2 -1770.699} C_VEL
LIN {X 0,Y 580.256,Z 262.522,A -85,B 0,C 180,E1 -1773.673,E2 -1773.673} C_VEL
LIN {X 0,Y 580.266,Z 262.51,A -85,B 0,C 180,E1 -1776.441,E2 -1776.441} C_VEL
LIN {X 0,Y 580.268,Z 262.517,A -85,B 0,C 180,E1 -1779.437,E2 -1779.437} C_VEL
LIN {X 0,Y 580.253,Z 262.521,A -85,B 0,C 180,E1 -1781.644,E2 -1781.644} C_VEL
LIN {X 0,Y 580.256,Z 262.519,A -85,B 0,C 180,E1 -1783.824,E2 -1783.824} C_VEL
LIN {X 0,Y 580.312,Z 262.509,A -85,B 0,C 180,E1 -1785.982,E2 -1785.982} C_VEL
LIN {X 0,Y 580.307,Z 262.505,A -85,B 0,C 180,E1 -1788.827,E2 -1788.827} C_VEL
LIN {X 0,Y 580.31,Z 262.514,A -85,B 0,C 180,E1 -1791.643,E2 -1791.643} C_VEL
LIN {X 0,Y 580.282,Z 262.513,A -85,B 0,C 180,E1 -1793.742,E2 -1793.742} C_VEL
LIN {X 0,Y 580.271,Z 262.515,A -85,B 0,C 180,E1 -1795.832,E2 -1795.832} C_VEL
LIN {X 0,Y 580.344,Z 262.504,A -85,B 0,C 180,E1 -1797.918,E2 -1797.918} C_VEL
LIN {X 0,Y 580.347,Z 262.5,A -85,B 0,C 180,E1 -1800.693,E2 -1800.693} C_VEL
LIN {X 0,Y 580.283,Z 262.518,A -85,B 0,C 180,E1 -1803.471,E2 -1803.471} C_VEL
LIN {X 0,Y 580.33,Z 262.508,A -85,B 0,C 180,E1 -1805.559,E2 -1805.559} C_VEL
LIN {X 0,Y 580.326,Z 262.502,A -85,B 0,C 180,E1 -1808.356,E2 -1808.356} C_VEL
LIN {X 0,Y 580.301,Z 262.516,A -85,B 0,C 180,E1 -1811.191,E2 -1811.191} C_VEL
LIN {X 0,Y 580.318,Z 262.506,A -85,B 0,C 180,E1 -1814.017,E2 -1814.017} C_VEL
LIN {X 0,Y 580.313,Z 262.51,A -85,B 0,C 180,E1 -1816.913,E2 -1816.913} C_VEL
LIN {X 0,Y 580.287,Z 262.51,A -85,B 0,C 180,E1 -1819.823,E2 -1819.823} C_VEL
LIN {X 0,Y 580.27,Z 262.511,A -85,B 0,C 180,E1 -1822.052,E2 -1822.052} C_VEL
LIN {X 0,Y 580.306,Z 262.517,A -85,B 0,C 180,E1 -1825.079,E2 -1825.079} C_VEL
LIN {X 0,Y 580.297,Z 262.507,A -85,B 0,C 180,E1 -1828.185,E2 -1828.185} C_VEL
LIN {X 0,Y 580.284,Z 262.514,A -85,B 0,C 180,E1 -1830.694,E2 -1830.694} C_VEL
LIN {X 0,Y 580.301,Z 262.512,A -85,B 0,C 180,E1 -1833.316,E2 -1833.316} C_VEL
LIN {X 0,Y 580.271,Z 262.51,A -85,B 0,C 180,E1 -1835.76,E2 -1835.76} C_VEL
LIN {X 0,Y 580.289,Z 262.509,A -85,B 0,C 180,E1 -1838.146,E2 -1838.146} C_VEL
LIN {X 0,Y 580.299,Z 262.516,A -85,B 0,C 180,E1 -1840.843,E2 -1840.843} C_VEL
LIN {X 0,Y 580.278,Z 262.51,A -85,B 0,C 180,E1 -1843.658,E2 -1843.658} C_VEL
LIN {X 0,Y 580.284,Z 262.516,A -85,B 0,C 180,E1 -1846.608,E2 -1846.608} C_VEL
LIN {X 0,Y 580.298,Z 262.513,A -85,B 0,C 180,E1 -1849.157,E2 -1849.157} C_VEL
LIN {X 0,Y 580.289,Z 262.509,A -85,B 0,C 180,E1 -1851.927,E2 -1851.927} C_VEL
LIN {X 0,Y 580.252,Z 262.518,A -85,B 0,C 180,E1 -1854.453,E2 -1854.453} C_VEL
LIN {X 0,Y 580.288,Z 262.516,A -85,B 0,C 180,E1 -1856.975,E2 -1856.975} C_VEL
LIN {X 0,Y 580.296,Z 262.51,A -85,B 0,C 180,E1 -1859.425,E2 -1859.425} C_VEL
LIN {X 0,Y 580.329,Z 262.609,A -85,B 0,C 180,E1 -1862.259,E2 -1862.259} C_VEL
LIN {X 0,Y 582.195,Z 269.674,A -85,B 0,C 180,E1 -1862.978,E2 -1862.978} C_VEL
LIN {X 0,Y 581.902,Z 297.41,A -85,B 0,C 180,E1 -1865.377,E2 -1865.377} C_VEL
LIN {X 0,Y 581.767,Z 311.893,A -85,B 0,C 180,E1 -1866.614,E2 -1866.614} C_VEL
LIN {X 0,Y 582.717,Z 318.16,A -85,B 0,C 180,E1 -1866.748,E2 -1866.748} C_VEL
LIN {X 0,Y 582.136,Z 519.43,A -85,B 0,C 180,E1 -1869.367,E2 -1869.367} C_VEL
LIN {X 0,Y 582.05,Z 536.005,A -85,B 0,C 180,E1 -1869.733,E2 -1869.733} C_VEL
LIN {X 0,Y 581.824,Z 552.242,A -85,B 0,C 180,E1 -1870.232,E2 -1870.232} C_VEL
LIN {X 0,Y 581.6,Z 569.05,A -85,B 0,C 180,E1 -1870.91,E2 -1870.91} C_VEL
LIN {X 0,Y 581.414,Z 584.304,A -85,B 0,C 180,E1 -1871.683,E2 -1871.683} C_VEL
LIN {X 0,Y 581.161,Z 598.783,A -85,B 0,C 180,E1 -1872.566,E2 -1872.566} C_VEL
LIN {X 0,Y 580.977,Z 612.541,A -85,B 0,C 180,E1 -1873.575,E2 -1873.575} C_VEL
LIN {X 0,Y 580.742,Z 624.073,A -85,B 0,C 180,E1 -1874.56,E2 -1874.56} C_VEL
LIN {X 0,Y 580.589,Z 635.621,A -85,B 0,C 180,E1 -1875.699,E2 -1875.699} C_VEL
LIN {X 0,Y 580.412,Z 647.335,A -85,B 0,C 180,E1 -1877.055,E2 -1877.055} C_VEL
LIN {X 0,Y 580.315,Z 657.677,A -85,B 0,C 180,E1 -1878.474,E2 -1878.474} C_VEL
LIN {X 0,Y 580.219,Z 666.286,A -85,B 0,C 180,E1 -1879.885,E2 -1879.885} C_VEL
LIN {X 0,Y 580.164,Z 673.488,A -85,B 0,C 180,E1 -1881.291,E2 -1881.291} C_VEL
LIN {X 0,Y 580.119,Z 679.467,A -85,B 0,C 180,E1 -1882.692,E2 -1882.692} C_VEL
LIN {X 0,Y 580.111,Z 685.247,A -85,B 0,C 180,E1 -1884.438,E2 -1884.438} C_VEL
LIN {X 0,Y 580.086,Z 688.635,A -85,B 0,C 180,E1 -1885.831,E2 -1885.831} C_VEL
LIN {X 0,Y 580.031,Z 691.088,A -85,B 0,C 180,E1 -1887.222,E2 -1887.222} C_VEL
LIN {X 0,Y 580.04,Z 692.479,A -85,B 0,C 180,E1 -1888.612,E2 -1888.612} C_VEL
LIN {X 0,Y 580.033,Z 693,A -85,B 0,C 180,E1 -1890,E2 -1890} C_VEL
LIN {X 0,Y 580.04,Z 692.479,A -85,B 0,C 180,E1 -1891.389,E2 -1891.389} C_VEL
LIN {X 0,Y 580.031,Z 691.087,A -85,B 0,C 180,E1 -1892.778,E2 -1892.778} C_VEL
LIN {X 0,Y 580.086,Z 688.635,A -85,B 0,C 180,E1 -1894.169,E2 -1894.169} C_VEL
LIN {X 0,Y 580.098,Z 684.187,A -85,B 0,C 180,E1 -1895.911,E2 -1895.911} C_VEL
LIN {X 0,Y 580.119,Z 679.468,A -85,B 0,C 180,E1 -1897.308,E2 -1897.308} C_VEL
LIN {X 0,Y 580.157,Z 671.856,A -85,B 0,C 180,E1 -1899.061,E2 -1899.061} C_VEL
LIN {X 0,Y 580.24,Z 663.249,A -85,B 0,C 180,E1 -1900.644,E2 -1900.644} C_VEL
LIN {X 0,Y 580.335,Z 653.971,A -85,B 0,C 180,E1 -1902.058,E2 -1902.058} C_VEL
LIN {X 0,Y 580.44,Z 644.423,A -85,B 0,C 180,E1 -1903.3,E2 -1903.3} C_VEL
LIN {X 0,Y 580.623,Z 632.93,A -85,B 0,C 180,E1 -1904.582,E2 -1904.582} C_VEL
LIN {X 0,Y 580.814,Z 621.141,A -85,B 0,C 180,E1 -1905.709,E2 -1905.709} C_VEL
LIN {X 0,Y 581.011,Z 607.876,A -85,B 0,C 180,E1 -1906.786,E2 -1906.786} C_VEL
LIN {X 0,Y 581.235,Z 593.429,A -85,B 0,C 180,E1 -1907.777,E2 -1907.777} C_VEL
LIN {X 0,Y 581.445,Z 579.27,A -85,B 0,C 180,E1 -1908.59,E2 -1908.59} C_VEL
LIN {X 0,Y 581.697,Z 564.006,A -85,B 0,C 180,E1 -1909.314,E2 -1909.314} C_VEL
LIN {X 0,Y 581.905,Z 548.34,A -85,B 0,C 180,E1 -1909.904,E2 -1909.904} C_VEL
LIN {X 0,Y 582.055,Z 532.345,A -85,B 0,C 180,E1 -1910.359,E2 -1910.359} C_VEL
LIN {X 0,Y 582.149,Z 516.424,A -85,B 0,C 180,E1 -1910.678,E2 -1910.678} C_VEL
LIN {X 0,Y 582.717,Z 317.341,A -85,B 0,C 180,E1 -1913.263,E2 -1913.263} C_VEL
LIN {X 0,Y 581.754,Z 311.946,A -85,B 0,C 180,E1 -1913.382,E2 -1913.382} C_VEL
LIN {X 0,Y 582.176,Z 277.505,A -85,B 0,C 180,E1 -1916.337,E2 -1916.337} C_VEL
LIN {X 0,Y 582.194,Z 269.668,A -85,B 0,C 180,E1 -1917.023,E2 -1917.023} C_VEL
LIN {X 0,Y 580.304,Z 262.514,A -85,B 0,C 180,E1 -1917.766,E2 -1917.766} C_VEL
LIN {X 0,Y 580.286,Z 262.513,A -85,B 0,C 180,E1 -1920.695,E2 -1920.695} C_VEL
LIN {X 0,Y 580.303,Z 262.517,A -85,B 0,C 180,E1 -1923.317,E2 -1923.317} C_VEL
LIN {X 0,Y 580.244,Z 262.517,A -85,B 0,C 180,E1 -1925.756,E2 -1925.756} C_VEL
LIN {X 0,Y 580.289,Z 262.51,A -85,B 0,C 180,E1 -1928.146,E2 -1928.146} C_VEL
LIN {X 0,Y 580.299,Z 262.513,A -85,B 0,C 180,E1 -1930.844,E2 -1930.844} C_VEL
LIN {X 0,Y 580.288,Z 262.511,A -85,B 0,C 180,E1 -1933.657,E2 -1933.657} C_VEL
LIN {X 0,Y 580.277,Z 262.513,A -85,B 0,C 180,E1 -1936.61,E2 -1936.61} C_VEL
LIN {X 0,Y 580.3,Z 262.515,A -85,B 0,C 180,E1 -1939.157,E2 -1939.157} C_VEL
LIN {X 0,Y 580.291,Z 262.507,A -85,B 0,C 180,E1 -1941.927,E2 -1941.927} C_VEL
LIN {X 0,Y 580.252,Z 262.516,A -85,B 0,C 180,E1 -1944.453,E2 -1944.453} C_VEL
LIN {X 0,Y 580.289,Z 262.516,A -85,B 0,C 180,E1 -1946.975,E2 -1946.975} C_VEL
LIN {X 0,Y 580.297,Z 262.51,A -85,B 0,C 180,E1 -1949.426,E2 -1949.426} C_VEL
LIN {X 0,Y 580.297,Z 262.505,A -85,B 0,C 180,E1 -1952.142,E2 -1952.142} C_VEL
LIN {X 0,Y 580.323,Z 262.507,A -85,B 0,C 180,E1 -1955.27,E2 -1955.27} C_VEL
LIN {X 0,Y 580.269,Z 262.509,A -85,B 0,C 180,E1 -1957.948,E2 -1957.948} C_VEL
LIN {X 0,Y 580.295,Z 262.514,A -85,B 0,C 180,E1 -1960.914,E2 -1960.914} C_VEL
LIN {X 0,Y 580.267,Z 262.509,A -85,B 0,C 180,E1 -1963.826,E2 -1963.826} C_VEL
LIN {X 0,Y 580.27,Z 262.52,A -85,B 0,C 180,E1 -1966.696,E2 -1966.696} C_VEL
LIN {X 0,Y 580.308,Z 262.509,A -85,B 0,C 180,E1 -1968.827,E2 -1968.827} C_VEL
LIN {X 0,Y 580.31,Z 262.506,A -85,B 0,C 180,E1 -1971.644,E2 -1971.644} C_VEL
LIN {X 0,Y 580.319,Z 262.513,A -85,B 0,C 180,E1 -1974.441,E2 -1974.441} C_VEL
LIN {X 0,Y 580.322,Z 262.505,A -85,B 0,C 180,E1 -1977.224,E2 -1977.224} C_VEL
LIN {X 0,Y 580.353,Z 262.504,A -85,B 0,C 180,E1 -1980,E2 -1980} C_VEL
LIN {X 0,Y 580.325,Z 262.507,A -85,B 0,C 180,E1 -1982.777,E2 -1982.777} C_VEL
LIN {X 0,Y 580.302,Z 262.507,A -85,B 0,C 180,E1 -1985.56,E2 -1985.56} C_VEL
LIN {X 0,Y 580.307,Z 262.513,A -85,B 0,C 180,E1 -1988.357,E2 -1988.357} C_VEL
LIN {X 0,Y 580.304,Z 262.507,A -85,B 0,C 180,E1 -1991.191,E2 -1991.191} C_VEL
LIN {X 0,Y 580.311,Z 262.51,A -85,B 0,C 180,E1 -1994.018,E2 -1994.018} C_VEL
LIN {X 0,Y 580.253,Z 262.514,A -85,B 0,C 180,E1 -1996.9,E2 -1996.9} C_VEL
LIN {X 0,Y 580.274,Z 262.512,A -85,B 0,C 180,E1 -1999.824,E2 -1999.824} C_VEL
LIN {X 0,Y 580.275,Z 262.511,A -85,B 0,C 180,E1 -2001.318,E2 -2001.318} C_VEL
LIN {X 0,Y 579.566,Z 262.606,A -85,B 0,C 180,E1 -2001.898,E2 -2001.898} C_VEL
LIN {X 0,Y 576.685,Z 262.961,A -85,B 0,C 180,E1 -2002.838,E2 -2002.838} C_VEL
LIN {X 0,Y 574.286,Z 263.259,A -85,B 0,C 180,E1 -2003.594,E2 -2003.594} C_VEL
LIN {X 0,Y 573.275,Z 263.389,A -85,B 0,C 180,E1 -2004.178,E2 -2004.178} C_VEL
LIN {X 0,Y 573.202,Z 263.393,A -85,B 0,C 180,E1 -2004.375,E2 -2004.375} C_VEL
LIN {X 0,Y 573.177,Z 263.394,A -85,B 0,C 180,E1 -2006.98,E2 -2006.98} C_VEL
LIN {X 0,Y 573.204,Z 263.393,A -85,B 0,C 180,E1 -2009.48,E2 -2009.48} C_VEL
LIN {X 0,Y 573.222,Z 263.396,A -85,B 0,C 180,E1 -2012.223,E2 -2012.223} C_VEL
LIN {X 0,Y 573.207,Z 263.391,A -85,B 0,C 180,E1 -2014.767,E2 -2014.767} C_VEL
LIN {X 0,Y 573.207,Z 263.4,A -85,B 0,C 180,E1 -2017.81,E2 -2017.81} C_VEL
LIN {X 0,Y 573.203,Z 263.393,A -85,B 0,C 180,E1 -2020.529,E2 -2020.529} C_VEL
LIN {X 0,Y 573.192,Z 263.396,A -85,B 0,C 180,E1 -2023.364,E2 -2023.364} C_VEL
LIN {X 0,Y 573.206,Z 263.394,A -85,B 0,C 180,E1 -2026.336,E2 -2026.336} C_VEL
LIN {X 0,Y 573.193,Z 263.395,A -85,B 0,C 180,E1 -2028.54,E2 -2028.54} C_VEL
LIN {X 0,Y 573.265,Z 263.495,A -85,B 0,C 180,E1 -2031.387,E2 -2031.387} C_VEL
LIN {X 0,Y 574.922,Z 270.293,A -85,B 0,C 180,E1 -2032.143,E2 -2032.143} C_VEL
LIN {X 0,Y 574.805,Z 282.941,A -85,B 0,C 180,E1 -2033.383,E2 -2033.383} C_VEL
LIN {X 0,Y 576.189,Z 290.695,A -85,B 0,C 180,E1 -2033.547,E2 -2033.547} C_VEL
LIN {X 0,Y 575.515,Z 489.518,A -85,B 0,C 180,E1 -2036.166,E2 -2036.166} C_VEL
LIN {X 0,Y 575.315,Z 506.016,A -85,B 0,C 180,E1 -2036.531,E2 -2036.531} C_VEL
LIN {X 0,Y 575.153,Z 521.405,A -85,B 0,C 180,E1 -2037.008,E2 -2037.008} C_VEL
LIN {X 0,Y 574.924,Z 536.882,A -85,B 0,C 180,E1 -2037.623,E2 -2037.623} C_VEL
LIN {X 0,Y 574.649,Z 551.913,A -85,B 0,C 180,E1 -2038.366,E2 -2038.366} C_VEL
LIN {X 0,Y 574.375,Z 566.98,A -85,B 0,C 180,E1 -2039.279,E2 -2039.279} C_VEL
LIN {X 0,Y 574.112,Z 579.432,A -85,B 0,C 180,E1 -2040.173,E2 -2040.173} C_VEL
LIN {X 0,Y 573.85,Z 592.513,A -85,B 0,C 180,E1 -2041.269,E2 -2041.269} C_VEL
LIN {X 0,Y 573.625,Z 604.573,A -85,B 0,C 180,E1 -2042.451,E2 -2042.451} C_VEL
LIN {X 0,Y 573.437,Z 616.392,A -85,B 0,C 180,E1 -2043.819,E2 -2043.819} C_VEL
LIN {X 0,Y 573.296,Z 625.904,A -85,B 0,C 180,E1 -2045.117,E2 -2045.117} C_VEL
LIN {X 0,Y 573.171,Z 634.655,A -85,B 0,C 180,E1 -2046.516,E2 -2046.516} C_VEL
LIN {X 0,Y 573.079,Z 642.614,A -85,B 0,C 180,E1 -2048.035,E2 -2048.035} C_VEL
LIN {X 0,Y 573.023,Z 649.049,A -85,B 0,C 180,E1 -2049.54,E2 -2049.54} C_VEL
LIN {X 0,Y 572.975,Z 653.456,A -85,B 0,C 180,E1 -2050.817,E2 -2050.817} C_VEL
LIN {X 0,Y 572.952,Z 657.116,A -85,B 0,C 180,E1 -2052.142,E2 -2052.142} C_VEL
LIN {X 0,Y 572.929,Z 660.114,A -85,B 0,C 180,E1 -2053.612,E2 -2053.612} C_VEL
LIN {X 0,Y 572.903,Z 662.043,A -85,B 0,C 180,E1 -2055.071,E2 -2055.071} C_VEL
LIN {X 0,Y 572.967,Z 662.89,A -85,B 0,C 180,E1 -2056.523,E2 -2056.523} C_VEL
LIN {X 0,Y 572.945,Z 662.796,A -85,B 0,C 180,E1 -2057.964,E2 -2057.964} C_VEL
LIN {X 0,Y 572.984,Z 661.621,A -85,B 0,C 180,E1 -2059.398,E2 -2059.398} C_VEL
LIN {X 0,Y 572.926,Z 659.537,A -85,B 0,C 180,E1 -2060.824,E2 -2060.824} C_VEL
LIN {X 0,Y 572.977,Z 656.365,A -85,B 0,C 180,E1 -2062.246,E2 -2062.246} C_VEL
LIN {X 0,Y 573.031,Z 652.214,A -85,B 0,C 180,E1 -2063.663,E2 -2063.663} C_VEL
LIN {X 0,Y 573.028,Z 646.939,A -85,B 0,C 180,E1 -2065.075,E2 -2065.075} C_VEL
LIN {X 0,Y 573.068,Z 640.51,A -85,B 0,C 180,E1 -2066.484,E2 -2066.484} C_VEL
LIN {X 0,Y 573.193,Z 632.843,A -85,B 0,C 180,E1 -2067.892,E2 -2067.892} C_VEL
LIN {X 0,Y 573.338,Z 622.445,A -85,B 0,C 180,E1 -2069.473,E2 -2069.473} C_VEL
LIN {X 0,Y 573.478,Z 611.39,A -85,B 0,C 180,E1 -2070.878,E2 -2070.878} C_VEL
LIN {X 0,Y 573.716,Z 599.996,A -85,B 0,C 180,E1 -2072.106,E2 -2072.106} C_VEL
LIN {X 0,Y 573.98,Z 586.639,A -85,B 0,C 180,E1 -2073.334,E2 -2073.334} C_VEL
LIN {X 0,Y 574.197,Z 573.129,A -85,B 0,C 180,E1 -2074.387,E2 -2074.387} C_VEL
LIN {X 0,Y 574.474,Z 558.384,A -85,B 0,C 180,E1 -2075.352,E2 -2075.352} C_VEL
LIN {X 0,Y 574.76,Z 543.899,A -85,B 0,C 180,E1 -2076.142,E2 -2076.142} C_VEL
LIN {X 0,Y 575.049,Z 527.902,A -85,B 0,C 180,E1 -2076.844,E2 -2076.844} C_VEL
LIN {X 0,Y 575.281,Z 511.868,A -85,B 0,C 180,E1 -2077.392,E2 -2077.392} C_VEL
LIN {X 0,Y 575.465,Z 494.85,A -85,B 0,C 180,E1 -2077.818,E2 -2077.818} C_VEL
LIN {X 0,Y 575.57,Z 477.231,A -85,B 0,C 180,E1 -2078.105,E2 -2078.105} C_VEL
LIN {X 0,Y 576.163,Z 290.802,A -85,B 0,C 180,E1 -2080.543,E2 -2080.543} C_VEL
LIN {X 0,Y 575.362,Z 285.617,A -85,B 0,C 180,E1 -2080.647,E2 -2080.647} C_VEL
LIN {X 0,Y 574.811,Z 282.723,A -85,B 0,C 180,E1 -2080.724,E2 -2080.724} C_VEL
LIN {X 0,Y 574.832,Z 269.674,A -85,B 0,C 180,E1 -2082.012,E2 -2082.012} C_VEL
LIN {X 0,Y 573.253,Z 263.393,A -85,B 0,C 180,E1 -2082.724,E2 -2082.724} C_VEL
LIN {X 0,Y 573.225,Z 263.392,A -85,B 0,C 180,E1 -2084.92,E2 -2084.92} C_VEL
LIN {X 0,Y 573.21,Z 263.395,A -85,B 0,C 180,E1 -2087.85,E2 -2087.85} C_VEL
LIN {X 0,Y 573.233,Z 263.396,A -85,B 0,C 180,E1 -2090.077,E2 -2090.077} C_VEL
LIN {X 0,Y 573.218,Z 263.398,A -85,B 0,C 180,E1 -2092.338,E2 -2092.338} C_VEL
LIN {X 0,Y 573.212,Z 263.391,A -85,B 0,C 180,E1 -2094.865,E2 -2094.865} C_VEL
LIN {X 0,Y 573.216,Z 263.394,A -85,B 0,C 180,E1 -2097.769,E2 -2097.769} C_VEL
LIN {X 0,Y 573.224,Z 263.399,A -85,B 0,C 180,E1 -2100.177,E2 -2100.177} C_VEL
LIN {X 0,Y 573.221,Z 263.392,A -85,B 0,C 180,E1 -2102.647,E2 -2102.647} C_VEL
LIN {X 0,Y 573.179,Z 263.393,A -85,B 0,C 180,E1 -2105.19,E2 -2105.19} C_VEL
LIN {X 0,Y 573.182,Z 263.4,A -85,B 0,C 180,E1 -2107.812,E2 -2107.812} C_VEL
LIN {X 0,Y 573.202,Z 263.394,A -85,B 0,C 180,E1 -2110.529,E2 -2110.529} C_VEL
LIN {X 0,Y 573.187,Z 263.394,A -85,B 0,C 180,E1 -2113.364,E2 -2113.364} C_VEL
LIN {X 0,Y 573.196,Z 263.395,A -85,B 0,C 180,E1 -2116.336,E2 -2116.336} C_VEL
LIN {X 0,Y 573.187,Z 263.395,A -85,B 0,C 180,E1 -2118.539,E2 -2118.539} C_VEL
LIN {X 0,Y 573.229,Z 263.388,A -85,B 0,C 180,E1 -2121.297,E2 -2121.297} C_VEL
LIN {X 0,Y 573.181,Z 263.397,A -85,B 0,C 180,E1 -2124.023,E2 -2124.023} C_VEL
LIN {X 0,Y 573.223,Z 263.389,A -85,B 0,C 180,E1 -2126.514,E2 -2126.514} C_VEL
LIN {X 0,Y 573.22,Z 263.39,A -85,B 0,C 180,E1 -2129.119,E2 -2129.119} C_VEL
LIN {X 0,Y 573.197,Z 263.398,A -85,B 0,C 180,E1 -2131.981,E2 -2131.981} C_VEL
LIN {X 0,Y 573.223,Z 263.388,A -85,B 0,C 180,E1 -2134.588,E2 -2134.588} C_VEL
LIN {X 0,Y 573.229,Z 263.396,A -85,B 0,C 180,E1 -2137.661,E2 -2137.661} C_VEL
LIN {X 0,Y 573.268,Z 263.383,A -85,B 0,C 180,E1 -2140.67,E2 -2140.67} C_VEL
LIN {X 0,Y 573.229,Z 263.397,A -85,B 0,C 180,E1 -2143.621,E2 -2143.621} C_VEL
LIN {X 0,Y 573.258,Z 263.39,A -85,B 0,C 180,E1 -2145.806,E2 -2145.806} C_VEL
LIN {X 0,Y 573.265,Z 263.382,A -85,B 0,C 180,E1 -2148.745,E2 -2148.745} C_VEL
LIN {X 0,Y 573.254,Z 263.395,A -85,B 0,C 180,E1 -2151.54,E2 -2151.54} C_VEL
LIN {X 0,Y 573.244,Z 263.391,A -85,B 0,C 180,E1 -2153.665,E2 -2153.665} C_VEL
LIN {X 0,Y 573.228,Z 263.393,A -85,B 0,C 180,E1 -2155.781,E2 -2155.781} C_VEL
LIN {X 0,Y 573.314,Z 263.38,A -85,B 0,C 180,E1 -2157.892,E2 -2157.892} C_VEL
LIN {X 0,Y 573.32,Z 263.375,A -85,B 0,C 180,E1 -2160.702,E2 -2160.702} C_VEL
LIN {X 0,Y 573.294,Z 263.381,A -85,B 0,C 180,E1 -2162.81,E2 -2162.81} C_VEL
LIN {X 0,Y 573.296,Z 263.383,A -85,B 0,C 180,E1 -2165.628,E2 -2165.628} C_VEL
LIN {X 0,Y 573.282,Z 263.38,A -85,B 0,C 180,E1 -2168.459,E2 -2168.459} C_VEL
LIN {X 0,Y 573.273,Z 263.392,A -85,B 0,C 180,E1 -2171.312,E2 -2171.312} C_VEL
LIN {X 0,Y 573.26,Z 263.384,A -85,B 0,C 180,E1 -2174.193,E2 -2174.193} C_VEL
LIN {X 0,Y 573.259,Z 263.393,A -85,B 0,C 180,E1 -2177.111,E2 -2177.111} C_VEL
LIN {X 0,Y 573.241,Z 263.387,A -85,B 0,C 180,E1 -2180.077,E2 -2180.077} C_VEL
LIN {X 0,Y 573.235,Z 263.387,A -85,B 0,C 180,E1 -2182.337,E2 -2182.337} C_VEL
LIN {X 0,Y 573.253,Z 263.391,A -85,B 0,C 180,E1 -2185.41,E2 -2185.41} C_VEL
LIN {X 0,Y 573.25,Z 263.385,A -85,B 0,C 180,E1 -2188.028,E2 -2188.028} C_VEL
LIN {X 0,Y 573.246,Z 263.386,A -85,B 0,C 180,E1 -2190.176,E2 -2190.176} C_VEL
LIN {X 0,Y 573.252,Z 263.389,A -85,B 0,C 180,E1 -2192.645,E2 -2192.645} C_VEL
LIN {X 0,Y 573.253,Z 263.391,A -85,B 0,C 180,E1 -2195.184,E2 -2195.184} C_VEL
LIN {X 0,Y 573.236,Z 263.387,A -85,B 0,C 180,E1 -2197.807,E2 -2197.807} C_VEL
LIN {X 0,Y 573.269,Z 263.387,A -85,B 0,C 180,E1 -2200.528,E2 -2200.528} C_VEL
LIN {X 0,Y 573.243,Z 263.387,A -85,B 0,C 180,E1 -2203.669,E2 -2203.669} C_VEL
LIN {X 0,Y 573.245,Z 263.393,A -85,B 0,C 180,E1 -2206.642,E2 -2206.642} C_VEL
LIN {X 0,Y 573.258,Z 263.386,A -85,B 0,C 180,E1 -2209.476,E2 -2209.476} C_VEL
LIN {X 0,Y 573.234,Z 263.389,A -85,B 0,C 180,E1 -2212.192,E2 -2212.192} C_VEL
LIN {X 0,Y 573.233,Z 263.391,A -85,B 0,C 180,E1 -2215.229,E2 -2215.229} C_VEL
LIN {X 0,Y 573.249,Z 263.387,A -85,B 0,C 180,E1 -2217.772,E2 -2217.772} C_VEL
LIN {X 0,Y 573.259,Z 263.394,A -85,B 0,C 180,E1 -2220.634,E2 -2220.634} C_VEL
LIN {X 0,Y 573.25,Z 263.402,A -85,B 0,C 180,E1 -2221.971,E2 -2221.971} C_VEL
LIN {X 0,Y 575.528,Z 271.309,A -85,B 0,C 180,E1 -2222.786,E2 -2222.786} C_VEL
LIN {X 0,Y 575.307,Z 292.965,A -85,B 0,C 180,E1 -2224.687,E2 -2224.687} C_VEL
LIN {X 0,Y 575.035,Z 311.957,A -85,B 0,C 180,E1 -2226.329,E2 -2226.329} C_VEL
LIN {X 0,Y 576.224,Z 319.185,A -85,B 0,C 180,E1 -2226.483,E2 -2226.483} C_VEL
LIN {X 0,Y 575.497,Z 519.43,A -85,B 0,C 180,E1 -2229.118,E2 -2229.118} C_VEL
LIN {X 0,Y 575.361,Z 536.006,A -85,B 0,C 180,E1 -2229.487,E2 -2229.487} C_VEL
LIN {X 0,Y 575.125,Z 552.243,A -85,B 0,C 180,E1 -2229.992,E2 -2229.992} C_VEL
LIN {X 0,Y 574.882,Z 568.197,A -85,B 0,C 180,E1 -2230.638,E2 -2230.638} C_VEL
LIN {X 0,Y 574.661,Z 582.719,A -85,B 0,C 180,E1 -2231.367,E2 -2231.367} C_VEL
LIN {X 0,Y 574.368,Z 597.651,A -85,B 0,C 180,E1 -2232.278,E2 -2232.278} C_VEL
LIN {X 0,Y 574.103,Z 611.383,A -85,B 0,C 180,E1 -2233.281,E2 -2233.281} C_VEL
LIN {X 0,Y 573.83,Z 624.071,A -85,B 0,C 180,E1 -2234.369,E2 -2234.369} C_VEL
LIN {X 0,Y 573.604,Z 636.28,A -85,B 0,C 180,E1 -2235.595,E2 -2235.595} C_VEL
LIN {X 0,Y 573.418,Z 647.336,A -85,B 0,C 180,E1 -2236.895,E2 -2236.895} C_VEL
LIN {X 0,Y 573.282,Z 657.673,A -85,B 0,C 180,E1 -2238.33,E2 -2238.33} C_VEL
LIN {X 0,Y 573.168,Z 666.285,A -85,B 0,C 180,E1 -2239.759,E2 -2239.759} C_VEL
LIN {X 0,Y 573.076,Z 673.489,A -85,B 0,C 180,E1 -2241.182,E2 -2241.182} C_VEL
